LIN {X 0,Y 298.467,Z 190.307,A -85,B 0,C 180,E1 -16356.676,E2 -16356.676} C_VEL
LIN {X 0,Y 298.543,Z 190.3,A -85,B 0,C 180,E1 -16360.757,E2 -16360.757} C_VEL
LIN {X 0,Y 298.576,Z 190.293,A -85,B 0,C 180,E1 -16364.994,E2 -16364.994} C_VEL
LIN {X 0,Y 298.576,Z 190.292,A -85,B 0,C 180,E1 -16369.146,E2 -16369.146} C_VEL
LIN {X 0,Y 298.726,Z 190.273,A -85,B 0,C 180,E1 -16371.885,E2 -16371.885} C_VEL
LIN {X 0,Y 298.643,Z 190.285,A -85,B 0,C 180,E1 -16374.599,E2 -16374.599} C_VEL
LIN {X 0,Y 298.901,Z 190.252,A -85,B 0,C 180,E1 -16378.653,E2 -16378.653} C_VEL
LIN {X 0,Y 298.909,Z 190.249,A -85,B 0,C 180,E1 -16381.348,E2 -16381.348} C_VEL
LIN {X 0,Y 298.644,Z 190.283,A -85,B 0,C 180,E1 -16385.402,E2 -16385.402} C_VEL
LIN {X 0,Y 298.715,Z 190.277,A -85,B 0,C 180,E1 -16388.116,E2 -16388.116} C_VEL
LIN {X 0,Y 298.531,Z 190.298,A -85,B 0,C 180,E1 -16392.233,E2 -16392.233} C_VEL
LIN {X 0,Y 298.57,Z 190.292,A -85,B 0,C 180,E1 -16395.195,E2 -16395.195} C_VEL
LIN {X 0,Y 298.524,Z 190.3,A -85,B 0,C 180,E1 -16399.245,E2 -16399.245} C_VEL
LIN {X 0,Y 298.443,Z 190.31,A -85,B 0,C 180,E1 -16403.599,E2 -16403.599} C_VEL
LIN {X 0,Y 298.473,Z 190.303,A -85,B 0,C 180,E1 -16406.576,E2 -16406.576} C_VEL
LIN {X 0,Y 298.409,Z 190.313,A -85,B 0,C 180,E1 -16409.643,E2 -16409.643} C_VEL
LIN {X 0,Y 298.385,Z 190.317,A -85,B 0,C 180,E1 -16412.802,E2 -16412.802} C_VEL
LIN {X 0,Y 298.434,Z 190.312,A -85,B 0,C 180,E1 -16416.808,E2 -16416.808} C_VEL
LIN {X 0,Y 298.379,Z 190.318,A -85,B 0,C 180,E1 -16421.089,E2 -16421.089} C_VEL
LIN {X 0,Y 298.393,Z 190.316,A -85,B 0,C 180,E1 -16423.105,E2 -16423.105} C_VEL
LIN {X 0,Y 298.365,Z 190.321,A -85,B 0,C 180,E1 -16426.917,E2 -16426.917} C_VEL
LIN {X 0,Y 298.344,Z 190.416,A -85,B 0,C 180,E1 -16428.923,E2 -16428.923} C_VEL
LIN {X 0,Y 298.563,Z 193.304,A -85,B 0,C 180,E1 -16432.266,E2 -16432.266} C_VEL
LIN {X 0,Y 298.418,Z 196.385,A -85,B 0,C 180,E1 -16435.584,E2 -16435.584} C_VEL
LIN {X 0,Y 298.069,Z 199.435,A -85,B 0,C 180,E1 -16438.755,E2 -16438.755} C_VEL
LIN {X 0,Y 297.76,Z 203.535,A -85,B 0,C 180,E1 -16442.859,E2 -16442.859} C_VEL
LIN {X 0,Y 302.246,Z 218.03,A -85,B 0,C 180,E1 -16443.997,E2 -16443.997} C_VEL
LIN {X 0,Y 305.227,Z 230.394,A -85,B 0,C 180,E1 -16445.154,E2 -16445.154} C_VEL
LIN {X 0,Y 307.051,Z 240.7,A -85,B 0,C 180,E1 -16446.285,E2 -16446.285} C_VEL
LIN {X 0,Y 307.3,Z 244.849,A -85,B 0,C 180,E1 -16446.769,E2 -16446.769} C_VEL
LIN {X 0,Y 305.731,Z 255.792,A -85,B 0,C 180,E1 -16448.066,E2 -16448.066} C_VEL
LIN {X 0,Y 303.889,Z 266.643,A -85,B 0,C 180,E1 -16449.703,E2 -16449.703} C_VEL
LIN {X 0,Y 302.308,Z 275.446,A -85,B 0,C 180,E1 -16451.358,E2 -16451.358} C_VEL
LIN {X 0,Y 300.868,Z 282.972,A -85,B 0,C 180,E1 -16453.093,E2 -16453.093} C_VEL
LIN {X 0,Y 299.745,Z 289.831,A -85,B 0,C 180,E1 -16455.054,E2 -16455.054} C_VEL
LIN {X 0,Y 298.55,Z 295.506,A -85,B 0,C 180,E1 -16457.077,E2 -16457.077} C_VEL
LIN {X 0,Y 297.731,Z 299.967,A -85,B 0,C 180,E1 -16459.115,E2 -16459.115} C_VEL
LIN {X 0,Y 297.363,Z 302.317,A -85,B 0,C 180,E1 -16460.477,E2 -16460.477} C_VEL
LIN {X 0,Y 297.061,Z 304.239,A -85,B 0,C 180,E1 -16461.839,E2 -16461.839} C_VEL
LIN {X 0,Y 296.697,Z 306.572,A -85,B 0,C 180,E1 -16464.203,E2 -16464.203} C_VEL
LIN {X 0,Y 296.631,Z 307.466,A -85,B 0,C 180,E1 -16465.923,E2 -16465.923} C_VEL
LIN {X 0,Y 296.574,Z 307.752,A -85,B 0,C 180,E1 -16467.283,E2 -16467.283} C_VEL
LIN {X 0,Y 296.52,Z 307.658,A -85,B 0,C 180,E1 -16468.641,E2 -16468.641} C_VEL
LIN {X 0,Y 296.528,Z 307.138,A -85,B 0,C 180,E1 -16469.999,E2 -16469.999} C_VEL
LIN {X 0,Y 296.769,Z 304.924,A -85,B 0,C 180,E1 -16472.714,E2 -16472.714} C_VEL
LIN {X 0,Y 297.167,Z 302.172,A -85,B 0,C 180,E1 -16474.747,E2 -16474.747} C_VEL
LIN {X 0,Y 297.771,Z 297.516,A -85,B 0,C 180,E1 -16477.205,E2 -16477.205} C_VEL
LIN {X 0,Y 298.63,Z 291.646,A -85,B 0,C 180,E1 -16479.48,E2 -16479.48} C_VEL
LIN {X 0,Y 299.615,Z 285.031,A -85,B 0,C 180,E1 -16481.499,E2 -16481.499} C_VEL
LIN {X 0,Y 301.103,Z 276.811,A -85,B 0,C 180,E1 -16483.496,E2 -16483.496} C_VEL
LIN {X 0,Y 302.376,Z 268.381,A -85,B 0,C 180,E1 -16485.156,E2 -16485.156} C_VEL
LIN {X 0,Y 303.801,Z 257.965,A -85,B 0,C 180,E1 -16486.806,E2 -16486.806} C_VEL
LIN {X 0,Y 305.133,Z 249.054,A -85,B 0,C 180,E1 -16487.94,E2 -16487.94} C_VEL
LIN {X 0,Y 305.873,Z 241.537,A -85,B 0,C 180,E1 -16488.762,E2 -16488.762} C_VEL
LIN {X 0,Y 304.35,Z 230.406,A -85,B 0,C 180,E1 -16489.929,E2 -16489.929} C_VEL
LIN {X 0,Y 301.664,Z 218.168,A -85,B 0,C 180,E1 -16491.009,E2 -16491.009} C_VEL
LIN {X 0,Y 298.079,Z 205.668,A -85,B 0,C 180,E1 -16491.918,E2 -16491.918} C_VEL
LIN {X 0,Y 297.554,Z 203.452,A -85,B 0,C 180,E1 -16492.052,E2 -16492.052} C_VEL
LIN {X 0,Y 297.889,Z 199.089,A -85,B 0,C 180,E1 -16496.294,E2 -16496.294} C_VEL
LIN {X 0,Y 298.135,Z 195.735,A -85,B 0,C 180,E1 -16499.669,E2 -16499.669} C_VEL
LIN {X 0,Y 298.333,Z 192.716,A -85,B 0,C 180,E1 -16502.804,E2 -16502.804} C_VEL
LIN {X 0,Y 298.394,Z 191.172,A -85,B 0,C 180,E1 -16504.477,E2 -16504.477} C_VEL
LIN {X 0,Y 298.365,Z 190.322,A -85,B 0,C 180,E1 -16506.073,E2 -16506.073} C_VEL
LIN {X 0,Y 298.39,Z 190.319,A -85,B 0,C 180,E1 -16509.485,E2 -16509.485} C_VEL
LIN {X 0,Y 298.415,Z 190.315,A -85,B 0,C 180,E1 -16513.106,E2 -16513.106} C_VEL
LIN {X 0,Y 298.455,Z 190.309,A -85,B 0,C 180,E1 -16516.929,E2 -16516.929} C_VEL
LIN {X 0,Y 298.414,Z 190.316,A -85,B 0,C 180,E1 -16520.997,E2 -16520.997} C_VEL
LIN {X 0,Y 298.402,Z 190.312,A -85,B 0,C 180,E1 -16523.927,E2 -16523.927} C_VEL
LIN {X 0,Y 298.375,Z 190.315,A -85,B 0,C 180,E1 -16527.981,E2 -16527.981} C_VEL
LIN {X 0,Y 298.442,Z 190.307,A -85,B 0,C 180,E1 -16531.902,E2 -16531.902} C_VEL
LIN {X 0,Y 298.471,Z 190.303,A -85,B 0,C 180,E1 -16534.922,E2 -16534.922} C_VEL
LIN {X 0,Y 298.45,Z 190.298,A -85,B 0,C 180,E1 -16537.866,E2 -16537.866} C_VEL
LIN {X 0,Y 298.534,Z 190.29,A -85,B 0,C 180,E1 -16540.756,E2 -16540.756} C_VEL
LIN {X 0,Y 298.568,Z 190.292,A -85,B 0,C 180,E1 -16544.993,E2 -16544.993} C_VEL
LIN {X 0,Y 298.598,Z 190.283,A -85,B 0,C 180,E1 -16549.146,E2 -16549.146} C_VEL
LIN {X 0,Y 298.754,Z 190.271,A -85,B 0,C 180,E1 -16551.885,E2 -16551.885} C_VEL
LIN {X 0,Y 298.766,Z 190.266,A -85,B 0,C 180,E1 -16553.042,E2 -16553.042} C_VEL
LIN {X 0,Y 298.162,Z 190.346,A -85,B 0,C 180,E1 -16554.166,E2 -16554.166} C_VEL
LIN {X 0,Y 295.36,Z 190.695,A -85,B 0,C 180,E1 -16555.997,E2 -16555.997} C_VEL
LIN {X 0,Y 292.958,Z 190.991,A -85,B 0,C 180,E1 -16557.483,E2 -16557.483} C_VEL
LIN {X 0,Y 291.935,Z 191.118,A -85,B 0,C 180,E1 -16558.634,E2 -16558.634} C_VEL
LIN {X 0,Y 291.858,Z 191.126,A -85,B 0,C 180,E1 -16559.023,E2 -16559.023} C_VEL
LIN {X 0,Y 291.866,Z 191.129,A -85,B 0,C 180,E1 -16561.379,E2 -16561.379} C_VEL
LIN {X 0,Y 291.609,Z 191.163,A -85,B 0,C 180,E1 -16565.532,E2 -16565.532} C_VEL
LIN {X 0,Y 291.682,Z 191.15,A -85,B 0,C 180,E1 -16568.312,E2 -16568.312} C_VEL
LIN {X 0,Y 291.495,Z 191.174,A -85,B 0,C 180,E1 -16572.532,E2 -16572.532} C_VEL
LIN {X 0,Y 291.485,Z 191.179,A -85,B 0,C 180,E1 -16575.38,E2 -16575.38} C_VEL
LIN {X 0,Y 291.461,Z 191.178,A -85,B 0,C 180,E1 -16579.894,E2 -16579.894} C_VEL
LIN {X 0,Y 291.406,Z 191.185,A -85,B 0,C 180,E1 -16584.205,E2 -16584.205} C_VEL
LIN {X 0,Y 291.401,Z 191.186,A -85,B 0,C 180,E1 -16587.274,E2 -16587.274} C_VEL
LIN {X 0,Y 291.316,Z 191.192,A -85,B 0,C 180,E1 -16590.439,E2 -16590.439} C_VEL
LIN {X 0,Y 291.324,Z 191.194,A -85,B 0,C 180,E1 -16593.701,E2 -16593.701} C_VEL
LIN {X 0,Y 291.38,Z 191.189,A -85,B 0,C 180,E1 -16597.262,E2 -16597.262} C_VEL
LIN {X 0,Y 291.385,Z 191.191,A -85,B 0,C 180,E1 -16600.634,E2 -16600.634} C_VEL
LIN {X 0,Y 291.484,Z 191.352,A -85,B 0,C 180,E1 -16604.365,E2 -16604.365} C_VEL
LIN {X 0,Y 292.156,Z 195.534,A -85,B 0,C 180,E1 -16608.221,E2 -16608.221} C_VEL
LIN {X 0,Y 292.726,Z 199.162,A -85,B 0,C 180,E1 -16611.379,E2 -16611.379} C_VEL
LIN {X 0,Y 292.864,Z 201.277,A -85,B 0,C 180,E1 -16613.139,E2 -16613.139} C_VEL
LIN {X 0,Y 292.676,Z 204.438,A -85,B 0,C 180,E1 -16615.65,E2 -16615.65} C_VEL
LIN {X 0,Y 291.929,Z 209.681,A -85,B 0,C 180,E1 -16619.635,E2 -16619.635} C_VEL
LIN {X 0,Y 291.017,Z 215.923,A -85,B 0,C 180,E1 -16624.237,E2 -16624.237} C_VEL
LIN {X 0,Y 290.861,Z 217.67,A -85,B 0,C 180,E1 -16625.405,E2 -16625.405} C_VEL
LIN {X 0,Y 293.908,Z 230.878,A -85,B 0,C 180,E1 -16626.259,E2 -16626.259} C_VEL
LIN {X 0,Y 296.022,Z 243.414,A -85,B 0,C 180,E1 -16627.287,E2 -16627.287} C_VEL
LIN {X 0,Y 297.282,Z 255.41,A -85,B 0,C 180,E1 -16628.483,E2 -16628.483} C_VEL
LIN {X 0,Y 297.664,Z 263.572,A -85,B 0,C 180,E1 -16629.441,E2 -16629.441} C_VEL
LIN {X 0,Y 295.955,Z 275.139,A -85,B 0,C 180,E1 -16630.945,E2 -16630.945} C_VEL
LIN {X 0,Y 294.469,Z 284.874,A -85,B 0,C 180,E1 -16632.547,E2 -16632.547} C_VEL
LIN {X 0,Y 293.094,Z 293.699,A -85,B 0,C 180,E1 -16634.352,E2 -16634.352} C_VEL
LIN {X 0,Y 291.791,Z 301.858,A -85,B 0,C 180,E1 -16636.42,E2 -16636.42} C_VEL
LIN {X 0,Y 290.885,Z 307.407,A -85,B 0,C 180,E1 -16638.151,E2 -16638.151} C_VEL
LIN {X 0,Y 290.171,Z 312.836,A -85,B 0,C 180,E1 -16640.241,E2 -16640.241} C_VEL
LIN {X 0,Y 289.724,Z 317.078,A -85,B 0,C 180,E1 -16642.334,E2 -16642.334} C_VEL
LIN {X 0,Y 289.474,Z 320.363,A -85,B 0,C 180,E1 -16644.514,E2 -16644.514} C_VEL
LIN {X 0,Y 289.431,Z 321.835,A -85,B 0,C 180,E1 -16645.824,E2 -16645.824} C_VEL
LIN {X 0,Y 289.438,Z 322.994,A -85,B 0,C 180,E1 -16647.218,E2 -16647.218} C_VEL
LIN {X 0,Y 289.415,Z 323.716,A -85,B 0,C 180,E1 -16648.61,E2 -16648.61} C_VEL
LIN {X 0,Y 289.435,Z 324.052,A -85,B 0,C 180,E1 -16650.001,E2 -16650.001} C_VEL
LIN {X 0,Y 289.407,Z 324,A -85,B 0,C 180,E1 -16651.392,E2 -16651.392} C_VEL
LIN {X 0,Y 289.429,Z 323.552,A -85,B 0,C 180,E1 -16652.784,E2 -16652.784} C_VEL
LIN {X 0,Y 289.476,Z 321.389,A -85,B 0,C 180,E1 -16655.574,E2 -16655.574} C_VEL
LIN {X 0,Y 289.728,Z 318.686,A -85,B 0,C 180,E1 -16657.667,E2 -16657.667} C_VEL
LIN {X 0,Y 290.255,Z 314.97,A -85,B 0,C 180,E1 -16659.759,E2 -16659.759} C_VEL
LIN {X 0,Y 291.005,Z 310.143,A -85,B 0,C 180,E1 -16661.846,E2 -16661.846} C_VEL
LIN {X 0,Y 292.152,Z 304.062,A -85,B 0,C 180,E1 -16663.919,E2 -16663.919} C_VEL
LIN {X 0,Y 293.63,Z 296.509,A -85,B 0,C 180,E1 -16665.977,E2 -16665.977} C_VEL
LIN {X 0,Y 295.102,Z 288.16,A -85,B 0,C 180,E1 -16667.811,E2 -16667.811} C_VEL
LIN {X 0,Y 296.864,Z 278.345,A -85,B 0,C 180,E1 -16669.535,E2 -16669.535} C_VEL
LIN {X 0,Y 298.763,Z 267.709,A -85,B 0,C 180,E1 -16671.022,E2 -16671.022} C_VEL
LIN {X 0,Y 299.201,Z 263.555,A -85,B 0,C 180,E1 -16671.531,E2 -16671.531} C_VEL
LIN {X 0,Y 298.318,Z 252.514,A -85,B 0,C 180,E1 -16672.845,E2 -16672.845} C_VEL
LIN {X 0,Y 296.83,Z 241.889,A -85,B 0,C 180,E1 -16673.919,E2 -16673.919} C_VEL
LIN {X 0,Y 294.402,Z 229.74,A -85,B 0,C 180,E1 -16674.961,E2 -16674.961} C_VEL
LIN {X 0,Y 291.231,Z 217.803,A -85,B 0,C 180,E1 -16675.81,E2 -16675.81} C_VEL
LIN {X 0,Y 291.171,Z 217.363,A -85,B 0,C 180,E1 -16675.83,E2 -16675.83} C_VEL
LIN {X 0,Y 292.11,Z 211.302,A -85,B 0,C 180,E1 -16680.346,E2 -16680.346} C_VEL
LIN {X 0,Y 292.873,Z 206.162,A -85,B 0,C 180,E1 -16684.326,E2 -16684.326} C_VEL
LIN {X 0,Y 293.02,Z 202.084,A -85,B 0,C 180,E1 -16687.675,E2 -16687.675} C_VEL
LIN {X 0,Y 292.72,Z 198.923,A -85,B 0,C 180,E1 -16690.407,E2 -16690.407} C_VEL
LIN {X 0,Y 292.016,Z 194.786,A -85,B 0,C 180,E1 -16694.26,E2 -16694.26} C_VEL
LIN {X 0,Y 291.354,Z 191.198,A -85,B 0,C 180,E1 -16698.017,E2 -16698.017} C_VEL
LIN {X 0,Y 291.342,Z 191.196,A -85,B 0,C 180,E1 -16701.157,E2 -16701.157} C_VEL
LIN {X 0,Y 291.35,Z 191.195,A -85,B 0,C 180,E1 -16704.625,E2 -16704.625} C_VEL
LIN {X 0,Y 291.353,Z 191.194,A -85,B 0,C 180,E1 -16707.949,E2 -16707.949} C_VEL
LIN {X 0,Y 291.354,Z 191.196,A -85,B 0,C 180,E1 -16711.156,E2 -16711.156} C_VEL
LIN {X 0,Y 291.401,Z 191.185,A -85,B 0,C 180,E1 -16714.271,E2 -16714.271} C_VEL
LIN {X 0,Y 291.408,Z 191.186,A -85,B 0,C 180,E1 -16717.302,E2 -16717.302} C_VEL
LIN {X 0,Y 291.49,Z 191.175,A -85,B 0,C 180,E1 -16720.273,E2 -16720.273} C_VEL
LIN {X 0,Y 291.526,Z 191.174,A -85,B 0,C 180,E1 -16724.634,E2 -16724.634} C_VEL
LIN {X 0,Y 291.52,Z 191.172,A -85,B 0,C 180,E1 -16728.88,E2 -16728.88} C_VEL
LIN {X 0,Y 291.673,Z 191.151,A -85,B 0,C 180,E1 -16731.688,E2 -16731.688} C_VEL
LIN {X 0,Y 291.613,Z 191.161,A -85,B 0,C 180,E1 -16734.468,E2 -16734.468} C_VEL
LIN {X 0,Y 291.868,Z 191.129,A -85,B 0,C 180,E1 -16738.621,E2 -16738.621} C_VEL
LIN {X 0,Y 291.876,Z 191.125,A -85,B 0,C 180,E1 -16741.38,E2 -16741.38} C_VEL
LIN {X 0,Y 291.614,Z 191.16,A -85,B 0,C 180,E1 -16745.532,E2 -16745.532} C_VEL
LIN {X 0,Y 291.664,Z 191.153,A -85,B 0,C 180,E1 -16748.313,E2 -16748.313} C_VEL
LIN {X 0,Y 291.499,Z 191.173,A -85,B 0,C 180,E1 -16752.533,E2 -16752.533} C_VEL
LIN {X 0,Y 291.524,Z 191.171,A -85,B 0,C 180,E1 -16755.378,E2 -16755.378} C_VEL
LIN {X 0,Y 291.438,Z 191.183,A -85,B 0,C 180,E1 -16759.876,E2 -16759.876} C_VEL
LIN {X 0,Y 291.385,Z 191.186,A -85,B 0,C 180,E1 -16764.207,E2 -16764.207} C_VEL
LIN {X 0,Y 291.408,Z 191.188,A -85,B 0,C 180,E1 -16767.273,E2 -16767.273} C_VEL
LIN {X 0,Y 291.326,Z 191.194,A -85,B 0,C 180,E1 -16770.439,E2 -16770.439} C_VEL
LIN {X 0,Y 291.334,Z 191.194,A -85,B 0,C 180,E1 -16773.7,E2 -16773.7} C_VEL
LIN {X 0,Y 291.362,Z 191.191,A -85,B 0,C 180,E1 -16777.254,E2 -16777.254} C_VEL
LIN {X 0,Y 291.324,Z 191.197,A -85,B 0,C 180,E1 -16780.645,E2 -16780.645} C_VEL
LIN {X 0,Y 291.285,Z 191.202,A -85,B 0,C 180,E1 -16784.404,E2 -16784.404} C_VEL
LIN {X 0,Y 291.289,Z 191.203,A -85,B 0,C 180,E1 -16788.413,E2 -16788.413} C_VEL
LIN {X 0,Y 291.533,Z 193.453,A -85,B 0,C 180,E1 -16791.189,E2 -16791.189} C_VEL
LIN {X 0,Y 291.548,Z 195.003,A -85,B 0,C 180,E1 -16792.942,E2 -16792.942} C_VEL
LIN {X 0,Y 291.283,Z 198.076,A -85,B 0,C 180,E1 -16796.295,E2 -16796.295} C_VEL
LIN {X 0,Y 290.967,Z 201.142,A -85,B 0,C 180,E1 -16799.522,E2 -16799.522} C_VEL
LIN {X 0,Y 290.749,Z 203.759,A -85,B 0,C 180,E1 -16802.196,E2 -16802.196} C_VEL
LIN {X 0,Y 294.319,Z 214.776,A -85,B 0,C 180,E1 -16803.063,E2 -16803.063} C_VEL
LIN {X 0,Y 297.609,Z 227.072,A -85,B 0,C 180,E1 -16804.212,E2 -16804.212} C_VEL
LIN {X 0,Y 299.924,Z 239.037,A -85,B 0,C 180,E1 -16805.521,E2 -16805.521} C_VEL
LIN {X 0,Y 300.63,Z 245.942,A -85,B 0,C 180,E1 -16806.353,E2 -16806.353} C_VEL
LIN {X 0,Y 298.943,Z 256.985,A -85,B 0,C 180,E1 -16807.723,E2 -16807.723} C_VEL
LIN {X 0,Y 297.212,Z 266.692,A -85,B 0,C 180,E1 -16809.226,E2 -16809.226} C_VEL
LIN {X 0,Y 295.583,Z 275.52,A -85,B 0,C 180,E1 -16810.918,E2 -16810.918} C_VEL
LIN {X 0,Y 294.067,Z 283.067,A -85,B 0,C 180,E1 -16812.69,E2 -16812.69} C_VEL
LIN {X 0,Y 292.837,Z 289.948,A -85,B 0,C 180,E1 -16814.693,E2 -16814.693} C_VEL
LIN {X 0,Y 291.61,Z 295.642,A -85,B 0,C 180,E1 -16816.764,E2 -16816.764} C_VEL
LIN {X 0,Y 290.733,Z 300.118,A -85,B 0,C 180,E1 -16818.849,E2 -16818.849} C_VEL
LIN {X 0,Y 290.332,Z 302.475,A -85,B 0,C 180,E1 -16820.244,E2 -16820.244} C_VEL
LIN {X 0,Y 290.007,Z 304.403,A -85,B 0,C 180,E1 -16821.639,E2 -16821.639} C_VEL
LIN {X 0,Y 289.597,Z 306.896,A -85,B 0,C 180,E1 -16824.272,E2 -16824.272} C_VEL
LIN {X 0,Y 289.55,Z 307.654,A -85,B 0,C 180,E1 -16825.824,E2 -16825.824} C_VEL
LIN {X 0,Y 289.503,Z 307.946,A -85,B 0,C 180,E1 -16827.216,E2 -16827.216} C_VEL
LIN {X 0,Y 289.441,Z 307.86,A -85,B 0,C 180,E1 -16828.608,E2 -16828.608} C_VEL
LIN {X 0,Y 289.445,Z 307.351,A -85,B 0,C 180,E1 -16829.999,E2 -16829.999} C_VEL
LIN {X 0,Y 289.697,Z 305.149,A -85,B 0,C 180,E1 -16832.78,E2 -16832.78} C_VEL
LIN {X 0,Y 290.119,Z 302.41,A -85,B 0,C 180,E1 -16834.862,E2 -16834.862} C_VEL
LIN {X 0,Y 290.631,Z 298.666,A -85,B 0,C 180,E1 -16836.943,E2 -16836.943} C_VEL
LIN {X 0,Y 291.344,Z 293.809,A -85,B 0,C 180,E1 -16839.019,E2 -16839.019} C_VEL
LIN {X 0,Y 292.281,Z 287.695,A -85,B 0,C 180,E1 -16841.089,E2 -16841.089} C_VEL
LIN {X 0,Y 293.672,Z 280.075,A -85,B 0,C 180,E1 -16843.139,E2 -16843.139} C_VEL
LIN {X 0,Y 295.257,Z 270.503,A -85,B 0,C 180,E1 -16845.177,E2 -16845.177} C_VEL
LIN {X 0,Y 296.76,Z 260.627,A -85,B 0,C 180,E1 -16846.862,E2 -16846.862} C_VEL
LIN {X 0,Y 298.153,Z 250.883,A -85,B 0,C 180,E1 -16848.197,E2 -16848.197} C_VEL
LIN {X 0,Y 299.049,Z 243.545,A -85,B 0,C 180,E1 -16849.029,E2 -16849.029} C_VEL
LIN {X 0,Y 298.349,Z 236.105,A -85,B 0,C 180,E1 -16849.87,E2 -16849.87} C_VEL
LIN {X 0,Y 296.394,Z 225.434,A -85,B 0,C 180,E1 -16850.941,E2 -16850.941} C_VEL
LIN {X 0,Y 293.199,Z 212.867,A -85,B 0,C 180,E1 -16852,E2 -16852} C_VEL
LIN {X 0,Y 290.55,Z 203.62,A -85,B 0,C 180,E1 -16852.658,E2 -16852.658} C_VEL
LIN {X 0,Y 290.859,Z 199.679,A -85,B 0,C 180,E1 -16856.615,E2 -16856.615} C_VEL
LIN {X 0,Y 291.162,Z 195.954,A -85,B 0,C 180,E1 -16860.454,E2 -16860.454} C_VEL
LIN {X 0,Y 291.334,Z 192.925,A -85,B 0,C 180,E1 -16863.696,E2 -16863.696} C_VEL
LIN {X 0,Y 291.305,Z 191.439,A -85,B 0,C 180,E1 -16865.378,E2 -16865.378} C_VEL
LIN {X 0,Y 291.343,Z 191.198,A -85,B 0,C 180,E1 -16867.244,E2 -16867.244} C_VEL
LIN {X 0,Y 291.323,Z 191.196,A -85,B 0,C 180,E1 -16870.639,E2 -16870.639} C_VEL
LIN {X 0,Y 291.331,Z 191.195,A -85,B 0,C 180,E1 -16874.389,E2 -16874.389} C_VEL
LIN {X 0,Y 291.372,Z 191.189,A -85,B 0,C 180,E1 -16878.388,E2 -16878.388} C_VEL
LIN {X 0,Y 291.362,Z 191.193,A -85,B 0,C 180,E1 -16881.159,E2 -16881.159} C_VEL
LIN {X 0,Y 291.345,Z 191.194,A -85,B 0,C 180,E1 -16884.623,E2 -16884.623} C_VEL
LIN {X 0,Y 291.352,Z 191.19,A -85,B 0,C 180,E1 -16887.948,E2 -16887.948} C_VEL
LIN {X 0,Y 291.361,Z 191.19,A -85,B 0,C 180,E1 -16891.156,E2 -16891.156} C_VEL
LIN {X 0,Y 291.398,Z 191.187,A -85,B 0,C 180,E1 -16894.27,E2 -16894.27} C_VEL
LIN {X 0,Y 291.401,Z 191.174,A -85,B 0,C 180,E1 -16897.301,E2 -16897.301} C_VEL
LIN {X 0,Y 291.482,Z 191.16,A -85,B 0,C 180,E1 -16900.271,E2 -16900.271} C_VEL
LIN {X 0,Y 291.517,Z 191.172,A -85,B 0,C 180,E1 -16904.633,E2 -16904.633} C_VEL
LIN {X 0,Y 291.533,Z 191.163,A -85,B 0,C 180,E1 -16908.88,E2 -16908.88} C_VEL
LIN {X 0,Y 291.702,Z 191.148,A -85,B 0,C 180,E1 -16911.688,E2 -16911.688} C_VEL
LIN {X 0,Y 291.609,Z 191.158,A -85,B 0,C 180,E1 -16914.468,E2 -16914.468} C_VEL
LIN {X 0,Y 291.86,Z 191.127,A -85,B 0,C 180,E1 -16918.62,E2 -16918.62} C_VEL
LIN {X 0,Y 291.858,Z 191.126,A -85,B 0,C 180,E1 -16919.023,E2 -16919.023} C_VEL
LIN {X 0,Y 291.164,Z 191.216,A -85,B 0,C 180,E1 -16920.176,E2 -16920.176} C_VEL
LIN {X 0,Y 288.155,Z 191.591,A -85,B 0,C 180,E1 -16922.047,E2 -16922.047} C_VEL
LIN {X 0,Y 285.627,Z 191.908,A -85,B 0,C 180,E1 -16923.567,E2 -16923.567} C_VEL
LIN {X 0,Y 284.588,Z 192.033,A -85,B 0,C 180,E1 -16924.749,E2 -16924.749} C_VEL
LIN {X 0,Y 284.529,Z 192.041,A -85,B 0,C 180,E1 -16925.15,E2 -16925.15} C_VEL
LIN {X 0,Y 284.672,Z 192.024,A -85,B 0,C 180,E1 -16927.09,E2 -16927.09} C_VEL
LIN {X 0,Y 284.542,Z 192.041,A -85,B 0,C 180,E1 -16929.956,E2 -16929.956} C_VEL
LIN {X 0,Y 284.445,Z 192.051,A -85,B 0,C 180,E1 -16934.304,E2 -16934.304} C_VEL
LIN {X 0,Y 284.398,Z 192.06,A -85,B 0,C 180,E1 -16938.739,E2 -16938.739} C_VEL
LIN {X 0,Y 284.335,Z 192.066,A -85,B 0,C 180,E1 -16941.762,E2 -16941.762} C_VEL
LIN {X 0,Y 284.34,Z 192.068,A -85,B 0,C 180,E1 -16944.846,E2 -16944.846} C_VEL
LIN {X 0,Y 284.31,Z 192.068,A -85,B 0,C 180,E1 -16948.013,E2 -16948.013} C_VEL
LIN {X 0,Y 284.274,Z 192.07,A -85,B 0,C 180,E1 -16951.277,E2 -16951.277} C_VEL
LIN {X 0,Y 284.343,Z 192.065,A -85,B 0,C 180,E1 -16955.356,E2 -16955.356} C_VEL
LIN {X 0,Y 284.313,Z 192.071,A -85,B 0,C 180,E1 -16958.169,E2 -16958.169} C_VEL
LIN {X 0,Y 284.327,Z 192.07,A -85,B 0,C 180,E1 -16962.143,E2 -16962.143} C_VEL
LIN {X 0,Y 284.381,Z 192.07,A -85,B 0,C 180,E1 -16963.786,E2 -16963.786} C_VEL
LIN {X 0,Y 285.063,Z 196.148,A -85,B 0,C 180,E1 -16967.699,E2 -16967.699} C_VEL
LIN {X 0,Y 285.517,Z 198.928,A -85,B 0,C 180,E1 -16970.214,E2 -16970.214} C_VEL
LIN {X 0,Y 285.824,Z 202.11,A -85,B 0,C 180,E1 -16972.961,E2 -16972.961} C_VEL
LIN {X 0,Y 285.667,Z 205.267,A -85,B 0,C 180,E1 -16975.543,E2 -16975.543} C_VEL
LIN {X 0,Y 284.838,Z 210.638,A -85,B 0,C 180,E1 -16979.721,E2 -16979.721} C_VEL
LIN {X 0,Y 284.074,Z 215.694,A -85,B 0,C 180,E1 -16983.559,E2 -16983.559} C_VEL
LIN {X 0,Y 283.873,Z 217.305,A -85,B 0,C 180,E1 -16984.77,E2 -16984.77} C_VEL
LIN {X 0,Y 287.066,Z 230.901,A -85,B 0,C 180,E1 -16985.697,E2 -16985.697} C_VEL
LIN {X 0,Y 289.187,Z 243.352,A -85,B 0,C 180,E1 -16986.755,E2 -16986.755} C_VEL
LIN {X 0,Y 290.454,Z 255.674,A -85,B 0,C 180,E1 -16988.024,E2 -16988.024} C_VEL
LIN {X 0,Y 290.924,Z 263.193,A -85,B 0,C 180,E1 -16988.943,E2 -16988.943} C_VEL
LIN {X 0,Y 289.25,Z 274.797,A -85,B 0,C 180,E1 -16990.485,E2 -16990.485} C_VEL
LIN {X 0,Y 287.883,Z 283.112,A -85,B 0,C 180,E1 -16991.857,E2 -16991.857} C_VEL
LIN {X 0,Y 286.548,Z 291.888,A -85,B 0,C 180,E1 -16993.619,E2 -16993.619} C_VEL
LIN {X 0,Y 285.081,Z 300.345,A -85,B 0,C 180,E1 -16995.73,E2 -16995.73} C_VEL
LIN {X 0,Y 283.883,Z 307.145,A -85,B 0,C 180,E1 -16997.854,E2 -16997.854} C_VEL
LIN {X 0,Y 283.149,Z 312.588,A -85,B 0,C 180,E1 -16999.996,E2 -16999.996} C_VEL
LIN {X 0,Y 282.678,Z 316.842,A -85,B 0,C 180,E1 -17002.142,E2 -17002.142} C_VEL
LIN {X 0,Y 282.369,Z 320.431,A -85,B 0,C 180,E1 -17004.61,E2 -17004.61} C_VEL
LIN {X 0,Y 282.345,Z 322.783,A -85,B 0,C 180,E1 -17007.148,E2 -17007.148} C_VEL
LIN {X 0,Y 282.338,Z 323.512,A -85,B 0,C 180,E1 -17008.575,E2 -17008.575} C_VEL
LIN {X 0,Y 282.354,Z 323.852,A -85,B 0,C 180,E1 -17010.001,E2 -17010.001} C_VEL
LIN {X 0,Y 282.33,Z 323.805,A -85,B 0,C 180,E1 -17011.427,E2 -17011.427} C_VEL
LIN {X 0,Y 282.335,Z 323.365,A -85,B 0,C 180,E1 -17012.854,E2 -17012.854} C_VEL
LIN {X 0,Y 282.385,Z 321.213,A -85,B 0,C 180,E1 -17015.714,E2 -17015.714} C_VEL
LIN {X 0,Y 282.685,Z 318.521,A -85,B 0,C 180,E1 -17017.86,E2 -17017.86} C_VEL
LIN {X 0,Y 283.22,Z 314.815,A -85,B 0,C 180,E1 -17020.003,E2 -17020.003} C_VEL
LIN {X 0,Y 284.031,Z 310,A -85,B 0,C 180,E1 -17022.141,E2 -17022.141} C_VEL
LIN {X 0,Y 285.239,Z 303.932,A -85,B 0,C 180,E1 -17024.264,E2 -17024.264} C_VEL
LIN {X 0,Y 286.757,Z 296.393,A -85,B 0,C 180,E1 -17026.37,E2 -17026.37} C_VEL
LIN {X 0,Y 288.258,Z 288.423,A -85,B 0,C 180,E1 -17028.173,E2 -17028.173} C_VEL
LIN {X 0,Y 290.152,Z 278.279,A -85,B 0,C 180,E1 -17030.006,E2 -17030.006} C_VEL
LIN {X 0,Y 292.147,Z 267.67,A -85,B 0,C 180,E1 -17031.521,E2 -17031.521} C_VEL
LIN {X 0,Y 292.393,Z 263.533,A -85,B 0,C 180,E1 -17032.059,E2 -17032.059} C_VEL
LIN {X 0,Y 291.611,Z 253.19,A -85,B 0,C 180,E1 -17033.332,E2 -17033.332} C_VEL
LIN {X 0,Y 289.912,Z 240.989,A -85,B 0,C 180,E1 -17034.611,E2 -17034.611} C_VEL
LIN {X 0,Y 287.221,Z 228.353,A -85,B 0,C 180,E1 -17035.72,E2 -17035.72} C_VEL
LIN {X 0,Y 284.247,Z 217.152,A -85,B 0,C 180,E1 -17036.545,E2 -17036.545} C_VEL
LIN {X 0,Y 285.064,Z 212.15,A -85,B 0,C 180,E1 -17040.357,E2 -17040.357} C_VEL
LIN {X 0,Y 285.845,Z 207.016,A -85,B 0,C 180,E1 -17044.435,E2 -17044.435} C_VEL
LIN {X 0,Y 286.032,Z 203.954,A -85,B 0,C 180,E1 -17047.01,E2 -17047.01} C_VEL
LIN {X 0,Y 285.743,Z 200.215,A -85,B 0,C 180,E1 -17050.319,E2 -17050.319} C_VEL
LIN {X 0,Y 285.166,Z 196.71,A -85,B 0,C 180,E1 -17053.633,E2 -17053.633} C_VEL
LIN {X 0,Y 284.386,Z 192.568,A -85,B 0,C 180,E1 -17057.846,E2 -17057.846} C_VEL
LIN {X 0,Y 284.284,Z 192.076,A -85,B 0,C 180,E1 -17058.601,E2 -17058.601} C_VEL
LIN {X 0,Y 284.311,Z 192.07,A -85,B 0,C 180,E1 -17062.277,E2 -17062.277} C_VEL
LIN {X 0,Y 284.297,Z 192.076,A -85,B 0,C 180,E1 -17065.349,E2 -17065.349} C_VEL
LIN {X 0,Y 284.275,Z 192.077,A -85,B 0,C 180,E1 -17068.723,E2 -17068.723} C_VEL
LIN {X 0,Y 284.378,Z 192.063,A -85,B 0,C 180,E1 -17072.828,E2 -17072.828} C_VEL
LIN {X 0,Y 284.37,Z 192.064,A -85,B 0,C 180,E1 -17076.707,E2 -17076.707} C_VEL
LIN {X 0,Y 284.418,Z 192.055,A -85,B 0,C 180,E1 -17079.873,E2 -17079.873} C_VEL
LIN {X 0,Y 284.463,Z 192.052,A -85,B 0,C 180,E1 -17084.469,E2 -17084.469} C_VEL
LIN {X 0,Y 284.472,Z 192.052,A -85,B 0,C 180,E1 -17088.601,E2 -17088.601} C_VEL
LIN {X 0,Y 284.624,Z 192.029,A -85,B 0,C 180,E1 -17091.48,E2 -17091.48} C_VEL
LIN {X 0,Y 284.583,Z 192.038,A -85,B 0,C 180,E1 -17094.331,E2 -17094.331} C_VEL
LIN {X 0,Y 284.834,Z 192.005,A -85,B 0,C 180,E1 -17098.586,E2 -17098.586} C_VEL
LIN {X 0,Y 284.842,Z 192.002,A -85,B 0,C 180,E1 -17101.414,E2 -17101.414} C_VEL
LIN {X 0,Y 284.624,Z 192.027,A -85,B 0,C 180,E1 -17106.681,E2 -17106.681} C_VEL
LIN {X 0,Y 284.498,Z 192.048,A -85,B 0,C 180,E1 -17109.958,E2 -17109.958} C_VEL
LIN {X 0,Y 284.462,Z 192.049,A -85,B 0,C 180,E1 -17114.304,E2 -17114.304} C_VEL
LIN {X 0,Y 284.411,Z 192.057,A -85,B 0,C 180,E1 -17117.25,E2 -17117.25} C_VEL
LIN {X 0,Y 284.366,Z 192.062,A -85,B 0,C 180,E1 -17120.244,E2 -17120.244} C_VEL
LIN {X 0,Y 284.355,Z 192.063,A -85,B 0,C 180,E1 -17123.876,E2 -17123.876} C_VEL
LIN {X 0,Y 284.384,Z 192.062,A -85,B 0,C 180,E1 -17127.174,E2 -17127.174} C_VEL
LIN {X 0,Y 284.284,Z 192.075,A -85,B 0,C 180,E1 -17131.276,E2 -17131.276} C_VEL
LIN {X 0,Y 284.331,Z 192.069,A -85,B 0,C 180,E1 -17135.349,E2 -17135.349} C_VEL
LIN {X 0,Y 284.299,Z 192.07,A -85,B 0,C 180,E1 -17138.172,E2 -17138.172} C_VEL
LIN {X 0,Y 284.262,Z 192.074,A -85,B 0,C 180,E1 -17142.126,E2 -17142.126} C_VEL
LIN {X 0,Y 284.232,Z 192.081,A -85,B 0,C 180,E1 -17146.187,E2 -17146.187} C_VEL
LIN {X 0,Y 284.236,Z 192.081,A -85,B 0,C 180,E1 -17148.12,E2 -17148.12} C_VEL
LIN {X 0,Y 284.447,Z 193.606,A -85,B 0,C 180,E1 -17150.031,E2 -17150.031} C_VEL
LIN {X 0,Y 284.532,Z 195.458,A -85,B 0,C 180,E1 -17152.225,E2 -17152.225} C_VEL
LIN {X 0,Y 284.337,Z 198.246,A -85,B 0,C 180,E1 -17155.356,E2 -17155.356} C_VEL
LIN {X 0,Y 284.016,Z 201.326,A -85,B 0,C 180,E1 -17158.693,E2 -17158.693} C_VEL
LIN {X 0,Y 283.777,Z 203.946,A -85,B 0,C 180,E1 -17161.463,E2 -17161.463} C_VEL
LIN {X 0,Y 285.69,Z 209.796,A -85,B 0,C 180,E1 -17161.939,E2 -17161.939} C_VEL
LIN {X 0,Y 289.595,Z 222.519,A -85,B 0,C 180,E1 -17163.109,E2 -17163.109} C_VEL
LIN {X 0,Y 292.212,Z 234.223,A -85,B 0,C 180,E1 -17164.348,E2 -17164.348} C_VEL
LIN {X 0,Y 293.963,Z 245.479,A -85,B 0,C 180,E1 -17165.733,E2 -17165.733} C_VEL
LIN {X 0,Y 292.96,Z 253.243,A -85,B 0,C 180,E1 -17166.683,E2 -17166.683} C_VEL
LIN {X 0,Y 291.162,Z 263.722,A -85,B 0,C 180,E1 -17168.216,E2 -17168.216} C_VEL
LIN {X 0,Y 289.564,Z 272.278,A -85,B 0,C 180,E1 -17169.766,E2 -17169.766} C_VEL
LIN {X 0,Y 287.927,Z 280.156,A -85,B 0,C 180,E1 -17171.5,E2 -17171.5} C_VEL
LIN {X 0,Y 286.256,Z 287.917,A -85,B 0,C 180,E1 -17173.625,E2 -17173.625} C_VEL
LIN {X 0,Y 285.141,Z 293.992,A -85,B 0,C 180,E1 -17175.731,E2 -17175.731} C_VEL
LIN {X 0,Y 283.984,Z 298.875,A -85,B 0,C 180,E1 -17177.857,E2 -17177.857} C_VEL
LIN {X 0,Y 283.314,Z 302.632,A -85,B 0,C 180,E1 -17180,E2 -17180} C_VEL
LIN {X 0,Y 282.953,Z 304.568,A -85,B 0,C 180,E1 -17181.429,E2 -17181.429} C_VEL
LIN {X 0,Y 282.682,Z 306.091,A -85,B 0,C 180,E1 -17182.859,E2 -17182.859} C_VEL
LIN {X 0,Y 282.526,Z 307.167,A -85,B 0,C 180,E1 -17184.289,E2 -17184.289} C_VEL
LIN {X 0,Y 282.433,Z 308.14,A -85,B 0,C 180,E1 -17187.147,E2 -17187.147} C_VEL
LIN {X 0,Y 282.364,Z 308.061,A -85,B 0,C 180,E1 -17188.573,E2 -17188.573} C_VEL
LIN {X 0,Y 282.365,Z 307.563,A -85,B 0,C 180,E1 -17189.999,E2 -17189.999} C_VEL
LIN {X 0,Y 282.628,Z 305.374,A -85,B 0,C 180,E1 -17192.85,E2 -17192.85} C_VEL
LIN {X 0,Y 283.071,Z 302.647,A -85,B 0,C 180,E1 -17194.984,E2 -17194.984} C_VEL
LIN {X 0,Y 283.577,Z 298.918,A -85,B 0,C 180,E1 -17197.117,E2 -17197.117} C_VEL
LIN {X 0,Y 284.334,Z 294.076,A -85,B 0,C 180,E1 -17199.244,E2 -17199.244} C_VEL
LIN {X 0,Y 285.315,Z 287.978,A -85,B 0,C 180,E1 -17201.363,E2 -17201.363} C_VEL
LIN {X 0,Y 286.79,Z 280.382,A -85,B 0,C 180,E1 -17203.46,E2 -17203.46} C_VEL
LIN {X 0,Y 288.432,Z 270.835,A -85,B 0,C 180,E1 -17205.545,E2 -17205.545} C_VEL
LIN {X 0,Y 289.979,Z 260.987,A -85,B 0,C 180,E1 -17207.269,E2 -17207.269} C_VEL
LIN {X 0,Y 291.425,Z 251.36,A -85,B 0,C 180,E1 -17208.622,E2 -17208.622} C_VEL
LIN {X 0,Y 292.355,Z 243.333,A -85,B 0,C 180,E1 -17209.558,E2 -17209.558} C_VEL
LIN {X 0,Y 290.773,Z 232.018,A -85,B 0,C 180,E1 -17210.851,E2 -17210.851} C_VEL
LIN {X 0,Y 288.376,Z 220.872,A -85,B 0,C 180,E1 -17211.938,E2 -17211.938} C_VEL
LIN {X 0,Y 284.796,Z 208.325,A -85,B 0,C 180,E1 -17212.961,E2 -17212.961} C_VEL
LIN {X 0,Y 283.549,Z 203.835,A -85,B 0,C 180,E1 -17213.278,E2 -17213.278} C_VEL
LIN {X 0,Y 283.823,Z 200.244,A -85,B 0,C 180,E1 -17216.945,E2 -17216.945} C_VEL
LIN {X 0,Y 284.1,Z 197.348,A -85,B 0,C 180,E1 -17220.022,E2 -17220.022} C_VEL
LIN {X 0,Y 284.289,Z 194.648,A -85,B 0,C 180,E1 -17222.944,E2 -17222.944} C_VEL
LIN {X 0,Y 284.295,Z 192.544,A -85,B 0,C 180,E1 -17225.334,E2 -17225.334} C_VEL
LIN {X 0,Y 284.259,Z 192.08,A -85,B 0,C 180,E1 -17226.393,E2 -17226.393} C_VEL
LIN {X 0,Y 284.296,Z 192.072,A -85,B 0,C 180,E1 -17229.992,E2 -17229.992} C_VEL
LIN {X 0,Y 284.283,Z 192.073,A -85,B 0,C 180,E1 -17234.197,E2 -17234.197} C_VEL
LIN {X 0,Y 284.324,Z 192.067,A -85,B 0,C 180,E1 -17238.133,E2 -17238.133} C_VEL
LIN {X 0,Y 284.324,Z 192.067,A -85,B 0,C 180,E1 -17242.271,E2 -17242.271} C_VEL
LIN {X 0,Y 284.292,Z 192.072,A -85,B 0,C 180,E1 -17245.348,E2 -17245.348} C_VEL
LIN {X 0,Y 284.276,Z 192.075,A -85,B 0,C 180,E1 -17248.723,E2 -17248.723} C_VEL
LIN {X 0,Y 284.376,Z 192.063,A -85,B 0,C 180,E1 -17252.825,E2 -17252.825} C_VEL
LIN {X 0,Y 284.362,Z 192.053,A -85,B 0,C 180,E1 -17256.706,E2 -17256.706} C_VEL
LIN {X 0,Y 284.41,Z 192.036,A -85,B 0,C 180,E1 -17259.872,E2 -17259.872} C_VEL
LIN {X 0,Y 284.455,Z 192.053,A -85,B 0,C 180,E1 -17264.468,E2 -17264.468} C_VEL
LIN {X 0,Y 284.495,Z 192.04,A -85,B 0,C 180,E1 -17268.601,E2 -17268.601} C_VEL
LIN {X 0,Y 284.651,Z 192.025,A -85,B 0,C 180,E1 -17271.481,E2 -17271.481} C_VEL
LIN {X 0,Y 284.58,Z 192.034,A -85,B 0,C 180,E1 -17274.33,E2 -17274.33} C_VEL
LIN {X 0,Y 284.827,Z 192.003,A -85,B 0,C 180,E1 -17278.586,E2 -17278.586} C_VEL
LIN {X 0,Y 284.833,Z 192.005,A -85,B 0,C 180,E1 -17281.414,E2 -17281.414} C_VEL
LIN {X 0,Y 284.529,Z 192.041,A -85,B 0,C 180,E1 -17285.15,E2 -17285.15} C_VEL
LIN {X 0,Y 283.918,Z 192.12,A -85,B 0,C 180,E1 -17286.333,E2 -17286.333} C_VEL
LIN {X 0,Y 281.044,Z 192.475,A -85,B 0,C 180,E1 -17288.259,E2 -17288.259} C_VEL
LIN {X 0,Y 278.564,Z 192.786,A -85,B 0,C 180,E1 -17289.824,E2 -17289.824} C_VEL
LIN {X 0,Y 277.496,Z 192.92,A -85,B 0,C 180,E1 -17291.039,E2 -17291.039} C_VEL
LIN {X 0,Y 277.409,Z 192.929,A -85,B 0,C 180,E1 -17291.45,E2 -17291.45} C_VEL
LIN {X 0,Y 277.393,Z 192.932,A -85,B 0,C 180,E1 -17295.704,E2 -17295.704} C_VEL
LIN {X 0,Y 277.352,Z 192.936,A -85,B 0,C 180,E1 -17300.367,E2 -17300.367} C_VEL
LIN {X 0,Y 277.312,Z 192.94,A -85,B 0,C 180,E1 -17304.178,E2 -17304.178} C_VEL
LIN {X 0,Y 277.305,Z 192.941,A -85,B 0,C 180,E1 -17307.507,E2 -17307.507} C_VEL
LIN {X 0,Y 277.253,Z 192.942,A -85,B 0,C 180,E1 -17310.484,E2 -17310.484} C_VEL
LIN {X 0,Y 277.235,Z 192.949,A -85,B 0,C 180,E1 -17313.897,E2 -17313.897} C_VEL
LIN {X 0,Y 277.268,Z 192.946,A -85,B 0,C 180,E1 -17317.469,E2 -17317.469} C_VEL
LIN {X 0,Y 277.25,Z 192.95,A -85,B 0,C 180,E1 -17321.229,E2 -17321.229} C_VEL
LIN {X 0,Y 277.342,Z 193.015,A -85,B 0,C 180,E1 -17323.422,E2 -17323.422} C_VEL
LIN {X 0,Y 277.976,Z 196.793,A -85,B 0,C 180,E1 -17327.155,E2 -17327.155} C_VEL
LIN {X 0,Y 278.585,Z 200.823,A -85,B 0,C 180,E1 -17330.904,E2 -17330.904} C_VEL
LIN {X 0,Y 278.777,Z 204.123,A -85,B 0,C 180,E1 -17333.777,E2 -17333.777} C_VEL
LIN {X 0,Y 278.432,Z 207.309,A -85,B 0,C 180,E1 -17336.404,E2 -17336.404} C_VEL
LIN {X 0,Y 277.606,Z 212.36,A -85,B 0,C 180,E1 -17340.421,E2 -17340.421} C_VEL
LIN {X 0,Y 276.884,Z 217.101,A -85,B 0,C 180,E1 -17344.113,E2 -17344.113} C_VEL
LIN {X 0,Y 280.195,Z 230.818,A -85,B 0,C 180,E1 -17345.095,E2 -17345.095} C_VEL
LIN {X 0,Y 282.349,Z 243.629,A -85,B 0,C 180,E1 -17346.224,E2 -17346.224} C_VEL
LIN {X 0,Y 283.545,Z 254.802,A -85,B 0,C 180,E1 -17347.413,E2 -17347.413} C_VEL
LIN {X 0,Y 284.12,Z 264.251,A -85,B 0,C 180,E1 -17348.604,E2 -17348.604} C_VEL
LIN {X 0,Y 282.551,Z 274.452,A -85,B 0,C 180,E1 -17350.003,E2 -17350.003} C_VEL
LIN {X 0,Y 281.11,Z 282.848,A -85,B 0,C 180,E1 -17351.415,E2 -17351.415} C_VEL
LIN {X 0,Y 279.725,Z 291.588,A -85,B 0,C 180,E1 -17353.208,E2 -17353.208} C_VEL
LIN {X 0,Y 278.438,Z 298.797,A -85,B 0,C 180,E1 -17355.008,E2 -17355.008} C_VEL
LIN {X 0,Y 277.086,Z 305.869,A -85,B 0,C 180,E1 -17357.179,E2 -17357.179} C_VEL
LIN {X 0,Y 276.139,Z 312.34,A -85,B 0,C 180,E1 -17359.739,E2 -17359.739} C_VEL
LIN {X 0,Y 275.605,Z 316.605,A -85,B 0,C 180,E1 -17361.939,E2 -17361.939} C_VEL
LIN {X 0,Y 275.302,Z 319.8,A -85,B 0,C 180,E1 -17364.141,E2 -17364.141} C_VEL
LIN {X 0,Y 275.248,Z 321.394,A -85,B 0,C 180,E1 -17365.608,E2 -17365.608} C_VEL
LIN {X 0,Y 275.255,Z 322.572,A -85,B 0,C 180,E1 -17367.074,E2 -17367.074} C_VEL
LIN {X 0,Y 275.262,Z 323.307,A -85,B 0,C 180,E1 -17368.538,E2 -17368.538} C_VEL
LIN {X 0,Y 275.276,Z 323.653,A -85,B 0,C 180,E1 -17370.001,E2 -17370.001} C_VEL
LIN {X 0,Y 275.255,Z 323.611,A -85,B 0,C 180,E1 -17371.464,E2 -17371.464} C_VEL
LIN {X 0,Y 275.244,Z 323.177,A -85,B 0,C 180,E1 -17372.928,E2 -17372.928} C_VEL
LIN {X 0,Y 275.299,Z 321.037,A -85,B 0,C 180,E1 -17375.861,E2 -17375.861} C_VEL
LIN {X 0,Y 275.616,Z 318.355,A -85,B 0,C 180,E1 -17378.062,E2 -17378.062} C_VEL
LIN {X 0,Y 276.208,Z 314.661,A -85,B 0,C 180,E1 -17380.26,E2 -17380.26} C_VEL
LIN {X 0,Y 277.047,Z 309.857,A -85,B 0,C 180,E1 -17382.452,E2 -17382.452} C_VEL
LIN {X 0,Y 278.609,Z 302.684,A -85,B 0,C 180,E1 -17384.984,E2 -17384.984} C_VEL
LIN {X 0,Y 280.238,Z 294.852,A -85,B 0,C 180,E1 -17387.138,E2 -17387.138} C_VEL
LIN {X 0,Y 281.785,Z 286.87,A -85,B 0,C 180,E1 -17388.919,E2 -17388.919} C_VEL
LIN {X 0,Y 283.699,Z 277.143,A -85,B 0,C 180,E1 -17390.671,E2 -17390.671} C_VEL
LIN {X 0,Y 285.701,Z 266.338,A -85,B 0,C 180,E1 -17392.222,E2 -17392.222} C_VEL
LIN {X 0,Y 285.192,Z 256.761,A -85,B 0,C 180,E1 -17393.495,E2 -17393.495} C_VEL
LIN {X 0,Y 283.928,Z 246.122,A -85,B 0,C 180,E1 -17394.723,E2 -17394.723} C_VEL
LIN {X 0,Y 281.673,Z 233.669,A -85,B 0,C 180,E1 -17395.941,E2 -17395.941} C_VEL
LIN {X 0,Y 278.159,Z 220.165,A -85,B 0,C 180,E1 -17397.058,E2 -17397.058} C_VEL
LIN {X 0,Y 277.302,Z 216.932,A -85,B 0,C 180,E1 -17397.293,E2 -17397.293} C_VEL
LIN {X 0,Y 278.094,Z 212.533,A -85,B 0,C 180,E1 -17400.768,E2 -17400.768} C_VEL
LIN {X 0,Y 278.827,Z 207.894,A -85,B 0,C 180,E1 -17404.548,E2 -17404.548} C_VEL
LIN {X 0,Y 279.02,Z 204.833,A -85,B 0,C 180,E1 -17407.192,E2 -17407.192} C_VEL
LIN {X 0,Y 278.636,Z 200.713,A -85,B 0,C 180,E1 -17410.978,E2 -17410.978} C_VEL
LIN {X 0,Y 277.933,Z 196.693,A -85,B 0,C 180,E1 -17414.926,E2 -17414.926} C_VEL
LIN {X 0,Y 277.24,Z 192.954,A -85,B 0,C 180,E1 -17418.984,E2 -17418.984} C_VEL
LIN {X 0,Y 277.256,Z 192.949,A -85,B 0,C 180,E1 -17422.529,E2 -17422.529} C_VEL
LIN {X 0,Y 277.235,Z 192.953,A -85,B 0,C 180,E1 -17426.103,E2 -17426.103} C_VEL
LIN {X 0,Y 277.251,Z 192.952,A -85,B 0,C 180,E1 -17429.537,E2 -17429.537} C_VEL
LIN {X 0,Y 277.339,Z 192.94,A -85,B 0,C 180,E1 -17432.862,E2 -17432.862} C_VEL
LIN {X 0,Y 277.331,Z 192.938,A -85,B 0,C 180,E1 -17436.08,E2 -17436.08} C_VEL
LIN {X 0,Y 277.357,Z 192.938,A -85,B 0,C 180,E1 -17440.767,E2 -17440.767} C_VEL
LIN {X 0,Y 277.412,Z 192.928,A -85,B 0,C 180,E1 -17445.325,E2 -17445.325} C_VEL
LIN {X 0,Y 277.446,Z 192.923,A -85,B 0,C 180,E1 -17449.787,E2 -17449.787} C_VEL
LIN {X 0,Y 277.627,Z 192.903,A -85,B 0,C 180,E1 -17452.729,E2 -17452.729} C_VEL
LIN {X 0,Y 277.801,Z 192.882,A -85,B 0,C 180,E1 -17458.551,E2 -17458.551} C_VEL
LIN {X 0,Y 277.809,Z 192.878,A -85,B 0,C 180,E1 -17461.45,E2 -17461.45} C_VEL
LIN {X 0,Y 277.572,Z 192.906,A -85,B 0,C 180,E1 -17466.699,E2 -17466.699} C_VEL
LIN {X 0,Y 277.55,Z 192.91,A -85,B 0,C 180,E1 -17469.073,E2 -17469.073} C_VEL
LIN {X 0,Y 277.397,Z 192.93,A -85,B 0,C 180,E1 -17473.181,E2 -17473.181} C_VEL
LIN {X 0,Y 277.388,Z 192.932,A -85,B 0,C 180,E1 -17476.183,E2 -17476.183} C_VEL
LIN {X 0,Y 277.333,Z 192.938,A -85,B 0,C 180,E1 -17480.351,E2 -17480.351} C_VEL
LIN {X 0,Y 277.305,Z 192.94,A -85,B 0,C 180,E1 -17484.17,E2 -17484.17} C_VEL
LIN {X 0,Y 277.313,Z 192.943,A -85,B 0,C 180,E1 -17487.506,E2 -17487.506} C_VEL
LIN {X 0,Y 277.263,Z 192.946,A -85,B 0,C 180,E1 -17490.483,E2 -17490.483} C_VEL
LIN {X 0,Y 277.238,Z 192.95,A -85,B 0,C 180,E1 -17493.898,E2 -17493.898} C_VEL
LIN {X 0,Y 277.255,Z 192.948,A -85,B 0,C 180,E1 -17497.472,E2 -17497.472} C_VEL
LIN {X 0,Y 277.202,Z 192.955,A -85,B 0,C 180,E1 -17501.239,E2 -17501.239} C_VEL
LIN {X 0,Y 277.189,Z 192.959,A -85,B 0,C 180,E1 -17505.23,E2 -17505.23} C_VEL
LIN {X 0,Y 277.187,Z 192.959,A -85,B 0,C 180,E1 -17507.332,E2 -17507.332} C_VEL
LIN {X 0,Y 277.349,Z 194.328,A -85,B 0,C 180,E1 -17509.482,E2 -17509.482} C_VEL
LIN {X 0,Y 277.498,Z 196.848,A -85,B 0,C 180,E1 -17512.569,E2 -17512.569} C_VEL
LIN {X 0,Y 277.205,Z 199.966,A -85,B 0,C 180,E1 -17516.1,E2 -17516.1} C_VEL
LIN {X 0,Y 276.81,Z 203.997,A -85,B 0,C 180,E1 -17520.534,E2 -17520.534} C_VEL
LIN {X 0,Y 276.807,Z 204.171,A -85,B 0,C 180,E1 -17520.719,E2 -17520.719} C_VEL
LIN {X 0,Y 278.655,Z 209.899,A -85,B 0,C 180,E1 -17521.194,E2 -17521.194} C_VEL
LIN {X 0,Y 282.357,Z 221.611,A -85,B 0,C 180,E1 -17522.309,E2 -17522.309} C_VEL
LIN {X 0,Y 285.109,Z 233.013,A -85,B 0,C 180,E1 -17523.552,E2 -17523.552} C_VEL
LIN {X 0,Y 287.003,Z 244.285,A -85,B 0,C 180,E1 -17524.965,E2 -17524.965} C_VEL
LIN {X 0,Y 287.325,Z 247.732,A -85,B 0,C 180,E1 -17525.43,E2 -17525.43} C_VEL
LIN {X 0,Y 285.357,Z 259.371,A -85,B 0,C 180,E1 -17526.985,E2 -17526.985} C_VEL
LIN {X 0,Y 283.565,Z 268.742,A -85,B 0,C 180,E1 -17528.558,E2 -17528.558} C_VEL
LIN {X 0,Y 281.803,Z 277.274,A -85,B 0,C 180,E1 -17530.326,E2 -17530.326} C_VEL
LIN {X 0,Y 279.945,Z 285.554,A -85,B 0,C 180,E1 -17532.467,E2 -17532.467} C_VEL
LIN {X 0,Y 278.666,Z 292.212,A -85,B 0,C 180,E1 -17534.644,E2 -17534.644} C_VEL
LIN {X 0,Y 277.325,Z 297.523,A -85,B 0,C 180,E1 -17536.816,E2 -17536.816} C_VEL
LIN {X 0,Y 276.514,Z 301.655,A -85,B 0,C 180,E1 -17539.011,E2 -17539.011} C_VEL
LIN {X 0,Y 275.92,Z 304.732,A -85,B 0,C 180,E1 -17541.209,E2 -17541.209} C_VEL
LIN {X 0,Y 275.619,Z 306.262,A -85,B 0,C 180,E1 -17542.675,E2 -17542.675} C_VEL
LIN {X 0,Y 275.44,Z 307.455,A -85,B 0,C 180,E1 -17544.336,E2 -17544.336} C_VEL
LIN {X 0,Y 275.341,Z 308.335,A -85,B 0,C 180,E1 -17547.073,E2 -17547.073} C_VEL
LIN {X 0,Y 275.29,Z 308.262,A -85,B 0,C 180,E1 -17548.536,E2 -17548.536} C_VEL
LIN {X 0,Y 275.287,Z 307.776,A -85,B 0,C 180,E1 -17549.999,E2 -17549.999} C_VEL
LIN {X 0,Y 275.561,Z 305.598,A -85,B 0,C 180,E1 -17552.923,E2 -17552.923} C_VEL
LIN {X 0,Y 276.026,Z 302.884,A -85,B 0,C 180,E1 -17555.111,E2 -17555.111} C_VEL
LIN {X 0,Y 276.53,Z 299.17,A -85,B 0,C 180,E1 -17557.299,E2 -17557.299} C_VEL
LIN {X 0,Y 277.329,Z 294.342,A -85,B 0,C 180,E1 -17559.479,E2 -17559.479} C_VEL
LIN {X 0,Y 278.375,Z 288.259,A -85,B 0,C 180,E1 -17561.65,E2 -17561.65} C_VEL
LIN {X 0,Y 279.914,Z 280.686,A -85,B 0,C 180,E1 -17563.797,E2 -17563.797} C_VEL
LIN {X 0,Y 281.624,Z 271.166,A -85,B 0,C 180,E1 -17565.931,E2 -17565.931} C_VEL
LIN {X 0,Y 283.238,Z 261.346,A -85,B 0,C 180,E1 -17567.693,E2 -17567.693} C_VEL
LIN {X 0,Y 284.705,Z 251.871,A -85,B 0,C 180,E1 -17569.062,E2 -17569.062} C_VEL
LIN {X 0,Y 285.604,Z 244.333,A -85,B 0,C 180,E1 -17569.972,E2 -17569.972} C_VEL
LIN {X 0,Y 284.007,Z 232.844,A -85,B 0,C 180,E1 -17571.341,E2 -17571.341} C_VEL
LIN {X 0,Y 281.489,Z 221.379,A -85,B 0,C 180,E1 -17572.512,E2 -17572.512} C_VEL
LIN {X 0,Y 278.019,Z 208.989,A -85,B 0,C 180,E1 -17573.565,E2 -17573.565} C_VEL
LIN {X 0,Y 276.529,Z 204.03,A -85,B 0,C 180,E1 -17573.929,E2 -17573.929} C_VEL
LIN {X 0,Y 276.817,Z 200.847,A -85,B 0,C 180,E1 -17577.3,E2 -17577.3} C_VEL
LIN {X 0,Y 277.091,Z 197.898,A -85,B 0,C 180,E1 -17580.479,E2 -17580.479} C_VEL
LIN {X 0,Y 277.265,Z 194.875,A -85,B 0,C 180,E1 -17583.889,E2 -17583.889} C_VEL
LIN {X 0,Y 277.235,Z 193.254,A -85,B 0,C 180,E1 -17585.785,E2 -17585.785} C_VEL
LIN {X 0,Y 277.245,Z 192.952,A -85,B 0,C 180,E1 -17588.201,E2 -17588.201} C_VEL
LIN {X 0,Y 277.222,Z 192.953,A -85,B 0,C 180,E1 -17592.676,E2 -17592.676} C_VEL
LIN {X 0,Y 277.25,Z 192.95,A -85,B 0,C 180,E1 -17596.809,E2 -17596.809} C_VEL
LIN {X 0,Y 277.252,Z 192.949,A -85,B 0,C 180,E1 -17600.674,E2 -17600.674} C_VEL
LIN {X 0,Y 277.272,Z 192.946,A -85,B 0,C 180,E1 -17604.339,E2 -17604.339} C_VEL
LIN {X 0,Y 277.226,Z 192.949,A -85,B 0,C 180,E1 -17607.833,E2 -17607.833} C_VEL
LIN {X 0,Y 277.251,Z 192.948,A -85,B 0,C 180,E1 -17611.208,E2 -17611.208} C_VEL
LIN {X 0,Y 277.3,Z 192.943,A -85,B 0,C 180,E1 -17614.478,E2 -17614.478} C_VEL
LIN {X 0,Y 277.287,Z 192.93,A -85,B 0,C 180,E1 -17617.654,E2 -17617.654} C_VEL
LIN {X 0,Y 277.349,Z 192.922,A -85,B 0,C 180,E1 -17620.766,E2 -17620.766} C_VEL
LIN {X 0,Y 277.405,Z 192.928,A -85,B 0,C 180,E1 -17625.324,E2 -17625.324} C_VEL
LIN {X 0,Y 277.53,Z 192.908,A -85,B 0,C 180,E1 -17629.789,E2 -17629.789} C_VEL
LIN {X 0,Y 277.639,Z 192.899,A -85,B 0,C 180,E1 -17632.728,E2 -17632.728} C_VEL
LIN {X 0,Y 277.793,Z 192.879,A -85,B 0,C 180,E1 -17638.55,E2 -17638.55} C_VEL
LIN {X 0,Y 277.799,Z 192.881,A -85,B 0,C 180,E1 -17641.449,E2 -17641.449} C_VEL
LIN {X 0,Y 277.549,Z 192.913,A -85,B 0,C 180,E1 -17645.813,E2 -17645.813} C_VEL
LIN {X 0,Y 277.606,Z 192.906,A -85,B 0,C 180,E1 -17649.158,E2 -17649.158} C_VEL
LIN {X 0,Y 277.409,Z 192.929,A -85,B 0,C 180,E1 -17651.45,E2 -17651.45} C_VEL
LIN {X 0,Y 276.728,Z 193.018,A -85,B 0,C 180,E1 -17652.663,E2 -17652.663} C_VEL
LIN {X 0,Y 273.821,Z 193.378,A -85,B 0,C 180,E1 -17654.636,E2 -17654.636} C_VEL
LIN {X 0,Y 271.369,Z 193.681,A -85,B 0,C 180,E1 -17656.24,E2 -17656.24} C_VEL
LIN {X 0,Y 270.338,Z 193.812,A -85,B 0,C 180,E1 -17657.485,E2 -17657.485} C_VEL
LIN {X 0,Y 270.265,Z 193.817,A -85,B 0,C 180,E1 -17657.907,E2 -17657.907} C_VEL
LIN {X 0,Y 270.243,Z 193.824,A -85,B 0,C 180,E1 -17661.351,E2 -17661.351} C_VEL
LIN {X 0,Y 270.258,Z 193.821,A -85,B 0,C 180,E1 -17664.587,E2 -17664.587} C_VEL
LIN {X 0,Y 270.252,Z 193.819,A -85,B 0,C 180,E1 -17667.911,E2 -17667.911} C_VEL
LIN {X 0,Y 270.165,Z 193.826,A -85,B 0,C 180,E1 -17671.35,E2 -17671.35} C_VEL
LIN {X 0,Y 270.197,Z 193.83,A -85,B 0,C 180,E1 -17674.906,E2 -17674.906} C_VEL
LIN {X 0,Y 270.207,Z 193.828,A -85,B 0,C 180,E1 -17678.72,E2 -17678.72} C_VEL
LIN {X 0,Y 270.278,Z 193.859,A -85,B 0,C 180,E1 -17682.926,E2 -17682.926} C_VEL
LIN {X 0,Y 270.895,Z 197.422,A -85,B 0,C 180,E1 -17686.587,E2 -17686.587} C_VEL
LIN {X 0,Y 271.575,Z 201.956,A -85,B 0,C 180,E1 -17690.928,E2 -17690.928} C_VEL
LIN {X 0,Y 271.757,Z 204.835,A -85,B 0,C 180,E1 -17693.505,E2 -17693.505} C_VEL
LIN {X 0,Y 271.483,Z 207.688,A -85,B 0,C 180,E1 -17695.934,E2 -17695.934} C_VEL
LIN {X 0,Y 270.883,Z 211.27,A -85,B 0,C 180,E1 -17698.89,E2 -17698.89} C_VEL
LIN {X 0,Y 269.952,Z 216.893,A -85,B 0,C 180,E1 -17703.422,E2 -17703.422} C_VEL
LIN {X 0,Y 273.353,Z 231.124,A -85,B 0,C 180,E1 -17704.489,E2 -17704.489} C_VEL
LIN {X 0,Y 275.468,Z 242.986,A -85,B 0,C 180,E1 -17705.58,E2 -17705.58} C_VEL
LIN {X 0,Y 276.71,Z 254.473,A -85,B 0,C 180,E1 -17706.835,E2 -17706.835} C_VEL
LIN {X 0,Y 277.323,Z 265.308,A -85,B 0,C 180,E1 -17708.248,E2 -17708.248} C_VEL
LIN {X 0,Y 275.456,Z 276.356,A -85,B 0,C 180,E1 -17709.855,E2 -17709.855} C_VEL
LIN {X 0,Y 273.665,Z 286.406,A -85,B 0,C 180,E1 -17711.705,E2 -17711.705} C_VEL
LIN {X 0,Y 272.28,Z 294.321,A -85,B 0,C 180,E1 -17713.507,E2 -17713.507} C_VEL
LIN {X 0,Y 270.787,Z 302.262,A -85,B 0,C 180,E1 -17715.728,E2 -17715.728} C_VEL
LIN {X 0,Y 269.619,Z 308.602,A -85,B 0,C 180,E1 -17717.966,E2 -17717.966} C_VEL
LIN {X 0,Y 268.912,Z 313.652,A -85,B 0,C 180,E1 -17720.221,E2 -17720.221} C_VEL
LIN {X 0,Y 268.426,Z 317.562,A -85,B 0,C 180,E1 -17722.479,E2 -17722.479} C_VEL
LIN {X 0,Y 268.171,Z 320.493,A -85,B 0,C 180,E1 -17724.793,E2 -17724.793} C_VEL
LIN {X 0,Y 268.167,Z 322.36,A -85,B 0,C 180,E1 -17726.997,E2 -17726.997} C_VEL
LIN {X 0,Y 268.188,Z 323.103,A -85,B 0,C 180,E1 -17728.499,E2 -17728.499} C_VEL
LIN {X 0,Y 268.2,Z 323.453,A -85,B 0,C 180,E1 -17730.001,E2 -17730.001} C_VEL
LIN {X 0,Y 268.181,Z 323.416,A -85,B 0,C 180,E1 -17731.503,E2 -17731.503} C_VEL
LIN {X 0,Y 268.155,Z 322.989,A -85,B 0,C 180,E1 -17733.005,E2 -17733.005} C_VEL
LIN {X 0,Y 268.163,Z 321.613,A -85,B 0,C 180,E1 -17735.188,E2 -17735.188} C_VEL
LIN {X 0,Y 268.563,Z 318.19,A -85,B 0,C 180,E1 -17738.276,E2 -17738.276} C_VEL
LIN {X 0,Y 269.208,Z 314.507,A -85,B 0,C 180,E1 -17740.53,E2 -17740.53} C_VEL
LIN {X 0,Y 270.082,Z 309.714,A -85,B 0,C 180,E1 -17742.779,E2 -17742.779} C_VEL
LIN {X 0,Y 271.748,Z 302.555,A -85,B 0,C 180,E1 -17745.372,E2 -17745.372} C_VEL
LIN {X 0,Y 273.444,Z 294.746,A -85,B 0,C 180,E1 -17747.577,E2 -17747.577} C_VEL
LIN {X 0,Y 275.059,Z 286.783,A -85,B 0,C 180,E1 -17749.4,E2 -17749.4} C_VEL
LIN {X 0,Y 277.053,Z 277.079,A -85,B 0,C 180,E1 -17751.19,E2 -17751.19} C_VEL
LIN {X 0,Y 278.926,Z 267.596,A -85,B 0,C 180,E1 -17752.596,E2 -17752.596} C_VEL
LIN {X 0,Y 278.503,Z 257.681,A -85,B 0,C 180,E1 -17753.979,E2 -17753.979} C_VEL
LIN {X 0,Y 277.207,Z 246.344,A -85,B 0,C 180,E1 -17755.348,E2 -17755.348} C_VEL
LIN {X 0,Y 275.046,Z 234.4,A -85,B 0,C 180,E1 -17756.579,E2 -17756.579} C_VEL
LIN {X 0,Y 271.665,Z 221.623,A -85,B 0,C 180,E1 -17757.71,E2 -17757.71} C_VEL
LIN {X 0,Y 270.41,Z 216.73,A -85,B 0,C 180,E1 -17758.082,E2 -17758.082} C_VEL
LIN {X 0,Y 271.101,Z 212.845,A -85,B 0,C 180,E1 -17761.229,E2 -17761.229} C_VEL
LIN {X 0,Y 271.821,Z 208.774,A -85,B 0,C 180,E1 -17764.666,E2 -17764.666} C_VEL
LIN {X 0,Y 271.962,Z 206.402,A -85,B 0,C 180,E1 -17766.765,E2 -17766.765} C_VEL
LIN {X 0,Y 271.846,Z 203.811,A -85,B 0,C 180,E1 -17769.142,E2 -17769.142} C_VEL
LIN {X 0,Y 271.433,Z 200.555,A -85,B 0,C 180,E1 -17772.312,E2 -17772.312} C_VEL
LIN {X 0,Y 270.659,Z 196.422,A -85,B 0,C 180,E1 -17776.637,E2 -17776.637} C_VEL
LIN {X 0,Y 270.204,Z 193.829,A -85,B 0,C 180,E1 -17779.685,E2 -17779.685} C_VEL
LIN {X 0,Y 270.215,Z 193.829,A -85,B 0,C 180,E1 -17783.73,E2 -17783.73} C_VEL
LIN {X 0,Y 270.19,Z 193.832,A -85,B 0,C 180,E1 -17786.891,E2 -17786.891} C_VEL
LIN {X 0,Y 270.181,Z 193.831,A -85,B 0,C 180,E1 -17790.381,E2 -17790.381} C_VEL
LIN {X 0,Y 270.25,Z 193.821,A -85,B 0,C 180,E1 -17793.763,E2 -17793.763} C_VEL
LIN {X 0,Y 270.24,Z 193.824,A -85,B 0,C 180,E1 -17797.04,E2 -17797.04} C_VEL
LIN {X 0,Y 270.314,Z 193.813,A -85,B 0,C 180,E1 -17800.246,E2 -17800.246} C_VEL
LIN {X 0,Y 270.381,Z 193.806,A -85,B 0,C 180,E1 -17804.934,E2 -17804.934} C_VEL
LIN {X 0,Y 270.398,Z 193.801,A -85,B 0,C 180,E1 -17809.518,E2 -17809.518} C_VEL
LIN {X 0,Y 270.585,Z 193.78,A -85,B 0,C 180,E1 -17812.538,E2 -17812.538} C_VEL
LIN {X 0,Y 270.767,Z 193.758,A -85,B 0,C 180,E1 -17818.513,E2 -17818.513} C_VEL
LIN {X 0,Y 270.775,Z 193.754,A -85,B 0,C 180,E1 -17821.488,E2 -17821.488} C_VEL
LIN {X 0,Y 270.528,Z 193.784,A -85,B 0,C 180,E1 -17826.71,E2 -17826.71} C_VEL
LIN {X 0,Y 270.511,Z 193.787,A -85,B 0,C 180,E1 -17829.176,E2 -17829.176} C_VEL
LIN {X 0,Y 270.34,Z 193.811,A -85,B 0,C 180,E1 -17833.531,E2 -17833.531} C_VEL
LIN {X 0,Y 270.32,Z 193.811,A -85,B 0,C 180,E1 -17836.618,E2 -17836.618} C_VEL
LIN {X 0,Y 270.28,Z 193.816,A -85,B 0,C 180,E1 -17840.602,E2 -17840.602} C_VEL
LIN {X 0,Y 270.262,Z 193.818,A -85,B 0,C 180,E1 -17844.587,E2 -17844.587} C_VEL
LIN {X 0,Y 270.26,Z 193.819,A -85,B 0,C 180,E1 -17847.91,E2 -17847.91} C_VEL
LIN {X 0,Y 270.175,Z 193.832,A -85,B 0,C 180,E1 -17851.35,E2 -17851.35} C_VEL
LIN {X 0,Y 270.192,Z 193.831,A -85,B 0,C 180,E1 -17854.908,E2 -17854.908} C_VEL
LIN {X 0,Y 270.191,Z 193.83,A -85,B 0,C 180,E1 -17858.712,E2 -17858.712} C_VEL
LIN {X 0,Y 270.159,Z 193.833,A -85,B 0,C 180,E1 -17863.251,E2 -17863.251} C_VEL
LIN {X 0,Y 270.174,Z 193.928,A -85,B 0,C 180,E1 -17867.445,E2 -17867.445} C_VEL
LIN {X 0,Y 270.455,Z 196.866,A -85,B 0,C 180,E1 -17871.223,E2 -17871.223} C_VEL
LIN {X 0,Y 270.42,Z 198.87,A -85,B 0,C 180,E1 -17873.676,E2 -17873.676} C_VEL
LIN {X 0,Y 270.094,Z 201.674,A -85,B 0,C 180,E1 -17876.879,E2 -17876.879} C_VEL
LIN {X 0,Y 269.812,Z 204.364,A -85,B 0,C 180,E1 -17879.906,E2 -17879.906} C_VEL
LIN {X 0,Y 274.79,Z 219.312,A -85,B 0,C 180,E1 -17881.335,E2 -17881.335} C_VEL
LIN {X 0,Y 277.736,Z 230.535,A -85,B 0,C 180,E1 -17882.567,E2 -17882.567} C_VEL
LIN {X 0,Y 279.654,Z 240.72,A -85,B 0,C 180,E1 -17883.831,E2 -17883.831} C_VEL
LIN {X 0,Y 280.648,Z 249.183,A -85,B 0,C 180,E1 -17885.009,E2 -17885.009} C_VEL
LIN {X 0,Y 278.618,Z 260.564,A -85,B 0,C 180,E1 -17886.592,E2 -17886.592} C_VEL
LIN {X 0,Y 276.555,Z 270.626,A -85,B 0,C 180,E1 -17888.378,E2 -17888.378} C_VEL
LIN {X 0,Y 274.752,Z 278.845,A -85,B 0,C 180,E1 -17890.189,E2 -17890.189} C_VEL
LIN {X 0,Y 272.914,Z 286.708,A -85,B 0,C 180,E1 -17892.331,E2 -17892.331} C_VEL
LIN {X 0,Y 271.794,Z 292.334,A -85,B 0,C 180,E1 -17894.246,E2 -17894.246} C_VEL
LIN {X 0,Y 270.397,Z 297.66,A -85,B 0,C 180,E1 -17896.472,E2 -17896.472} C_VEL
LIN {X 0,Y 269.513,Z 301.806,A -85,B 0,C 180,E1 -17898.721,E2 -17898.721} C_VEL
LIN {X 0,Y 268.876,Z 304.897,A -85,B 0,C 180,E1 -17900.977,E2 -17900.977} C_VEL
LIN {X 0,Y 268.553,Z 306.434,A -85,B 0,C 180,E1 -17902.481,E2 -17902.481} C_VEL
LIN {X 0,Y 268.36,Z 307.735,A -85,B 0,C 180,E1 -17904.374,E2 -17904.374} C_VEL
LIN {X 0,Y 268.252,Z 308.53,A -85,B 0,C 180,E1 -17906.996,E2 -17906.996} C_VEL
LIN {X 0,Y 268.217,Z 308.462,A -85,B 0,C 180,E1 -17908.498,E2 -17908.498} C_VEL
LIN {X 0,Y 268.21,Z 307.988,A -85,B 0,C 180,E1 -17909.999,E2 -17909.999} C_VEL
LIN {X 0,Y 268.496,Z 305.823,A -85,B 0,C 180,E1 -17913,E2 -17913} C_VEL
LIN {X 0,Y 268.961,Z 303.122,A -85,B 0,C 180,E1 -17915.246,E2 -17915.246} C_VEL
LIN {X 0,Y 269.673,Z 298.51,A -85,B 0,C 180,E1 -17917.971,E2 -17917.971} C_VEL
LIN {X 0,Y 270.674,Z 292.743,A -85,B 0,C 180,E1 -17920.47,E2 -17920.47} C_VEL
LIN {X 0,Y 271.899,Z 286.194,A -85,B 0,C 180,E1 -17922.69,E2 -17922.69} C_VEL
LIN {X 0,Y 273.61,Z 278.051,A -85,B 0,C 180,E1 -17924.882,E2 -17924.882} C_VEL
LIN {X 0,Y 275.154,Z 269.726,A -85,B 0,C 180,E1 -17926.697,E2 -17926.697} C_VEL
LIN {X 0,Y 276.843,Z 259.462,A -85,B 0,C 180,E1 -17928.499,E2 -17928.499} C_VEL
LIN {X 0,Y 278.241,Z 251.207,A -85,B 0,C 180,E1 -17929.675,E2 -17929.675} C_VEL
LIN {X 0,Y 278.885,Z 245.408,A -85,B 0,C 180,E1 -17930.397,E2 -17930.397} C_VEL
LIN {X 0,Y 277.512,Z 235.056,A -85,B 0,C 180,E1 -17931.694,E2 -17931.694} C_VEL
LIN {X 0,Y 274.904,Z 222.766,A -85,B 0,C 180,E1 -17933.021,E2 -17933.021} C_VEL
LIN {X 0,Y 271.395,Z 210.168,A -85,B 0,C 180,E1 -17934.163,E2 -17934.163} C_VEL
LIN {X 0,Y 269.493,Z 204.217,A -85,B 0,C 180,E1 -17934.659,E2 -17934.659} C_VEL
LIN {X 0,Y 269.829,Z 201.165,A -85,B 0,C 180,E1 -17937.955,E2 -17937.955} C_VEL
LIN {X 0,Y 270.111,Z 198.138,A -85,B 0,C 180,E1 -17941.354,E2 -17941.354} C_VEL
LIN {X 0,Y 270.222,Z 195.089,A -85,B 0,C 180,E1 -17944.898,E2 -17944.898} C_VEL
LIN {X 0,Y 270.15,Z 193.839,A -85,B 0,C 180,E1 -17946.747,E2 -17946.747} C_VEL
LIN {X 0,Y 270.167,Z 193.832,A -85,B 0,C 180,E1 -17950.562,E2 -17950.562} C_VEL
LIN {X 0,Y 270.177,Z 193.831,A -85,B 0,C 180,E1 -17954.609,E2 -17954.609} C_VEL
LIN {X 0,Y 270.253,Z 193.823,A -85,B 0,C 180,E1 -17958.945,E2 -17958.945} C_VEL
LIN {X 0,Y 270.219,Z 193.826,A -85,B 0,C 180,E1 -17963.258,E2 -17963.258} C_VEL
LIN {X 0,Y 270.185,Z 193.83,A -85,B 0,C 180,E1 -17966.889,E2 -17966.889} C_VEL
LIN {X 0,Y 270.178,Z 193.831,A -85,B 0,C 180,E1 -17970.38,E2 -17970.38} C_VEL
LIN {X 0,Y 270.247,Z 193.82,A -85,B 0,C 180,E1 -17973.762,E2 -17973.762} C_VEL
LIN {X 0,Y 270.232,Z 193.809,A -85,B 0,C 180,E1 -17977.038,E2 -17977.038} C_VEL
LIN {X 0,Y 270.306,Z 193.792,A -85,B 0,C 180,E1 -17980.244,E2 -17980.244} C_VEL
LIN {X 0,Y 270.374,Z 193.804,A -85,B 0,C 180,E1 -17984.933,E2 -17984.933} C_VEL
LIN {X 0,Y 270.472,Z 193.786,A -85,B 0,C 180,E1 -17989.52,E2 -17989.52} C_VEL
LIN {X 0,Y 270.597,Z 193.777,A -85,B 0,C 180,E1 -17992.538,E2 -17992.538} C_VEL
LIN {X 0,Y 270.759,Z 193.756,A -85,B 0,C 180,E1 -17998.512,E2 -17998.512} C_VEL
LIN {X 0,Y 270.766,Z 193.758,A -85,B 0,C 180,E1 -18001.487,E2 -18001.487} C_VEL
LIN {X 0,Y 270.585,Z 193.781,A -85,B 0,C 180,E1 -18007.462,E2 -18007.462} C_VEL
LIN {X 0,Y 270.418,Z 193.799,A -85,B 0,C 180,E1 -18010.482,E2 -18010.482} C_VEL
LIN {X 0,Y 270.359,Z 193.809,A -85,B 0,C 180,E1 -18015.067,E2 -18015.067} C_VEL
LIN {X 0,Y 270.265,Z 193.817,A -85,B 0,C 180,E1 -18017.907,E2 -18017.907} C_VEL
LIN {X 0,Y 269.61,Z 193.903,A -85,B 0,C 180,E1 -18019.151,E2 -18019.151} C_VEL
LIN {X 0,Y 266.715,Z 194.264,A -85,B 0,C 180,E1 -18021.176,E2 -18021.176} C_VEL
LIN {X 0,Y 264.268,Z 194.569,A -85,B 0,C 180,E1 -18022.823,E2 -18022.823} C_VEL
LIN {X 0,Y 263.254,Z 194.692,A -85,B 0,C 180,E1 -18024.102,E2 -18024.102} C_VEL
LIN {X 0,Y 263.192,Z 194.7,A -85,B 0,C 180,E1 -18024.535,E2 -18024.535} C_VEL
LIN {X 0,Y 263.16,Z 194.703,A -85,B 0,C 180,E1 -18028.732,E2 -18028.732} C_VEL
LIN {X 0,Y 263.115,Z 194.706,A -85,B 0,C 180,E1 -18032.291,E2 -18032.291} C_VEL
LIN {X 0,Y 263.17,Z 194.703,A -85,B 0,C 180,E1 -18035.981,E2 -18035.981} C_VEL
LIN {X 0,Y 263.145,Z 194.707,A -85,B 0,C 180,E1 -18039.865,E2 -18039.865} C_VEL
LIN {X 0,Y 263.271,Z 194.909,A -85,B 0,C 180,E1 -18042.639,E2 -18042.639} C_VEL
LIN {X 0,Y 263.852,Z 198.225,A -85,B 0,C 180,E1 -18046.174,E2 -18046.174} C_VEL
LIN {X 0,Y 264.469,Z 202.514,A -85,B 0,C 180,E1 -18050.412,E2 -18050.412} C_VEL
LIN {X 0,Y 264.719,Z 205.054,A -85,B 0,C 180,E1 -18052.794,E2 -18052.794} C_VEL
LIN {X 0,Y 264.551,Z 208.043,A -85,B 0,C 180,E1 -18055.441,E2 -18055.441} C_VEL
LIN {X 0,Y 263.631,Z 212.926,A -85,B 0,C 180,E1 -18059.572,E2 -18059.572} C_VEL
LIN {X 0,Y 263.001,Z 216.738,A -85,B 0,C 180,E1 -18062.708,E2 -18062.708} C_VEL
LIN {X 0,Y 266.272,Z 230.077,A -85,B 0,C 180,E1 -18063.732,E2 -18063.732} C_VEL
LIN {X 0,Y 268.271,Z 240.397,A -85,B 0,C 180,E1 -18064.695,E2 -18064.695} C_VEL
LIN {X 0,Y 269.776,Z 252.783,A -85,B 0,C 180,E1 -18066.061,E2 -18066.061} C_VEL
LIN {X 0,Y 270.522,Z 264.919,A -85,B 0,C 180,E1 -18067.672,E2 -18067.672} C_VEL
LIN {X 0,Y 269.205,Z 273.762,A -85,B 0,C 180,E1 -18068.966,E2 -18068.966} C_VEL
LIN {X 0,Y 267.269,Z 284.123,A -85,B 0,C 180,E1 -18070.813,E2 -18070.813} C_VEL
LIN {X 0,Y 265.74,Z 292.818,A -85,B 0,C 180,E1 -18072.768,E2 -18072.768} C_VEL
LIN {X 0,Y 264.151,Z 300.757,A -85,B 0,C 180,E1 -18074.967,E2 -18074.967} C_VEL
LIN {X 0,Y 263.004,Z 306.36,A -85,B 0,C 180,E1 -18076.873,E2 -18076.873} C_VEL
LIN {X 0,Y 262.081,Z 311.84,A -85,B 0,C 180,E1 -18079.183,E2 -18079.183} C_VEL
LIN {X 0,Y 261.507,Z 316.13,A -85,B 0,C 180,E1 -18081.501,E2 -18081.501} C_VEL
LIN {X 0,Y 261.155,Z 319.349,A -85,B 0,C 180,E1 -18083.822,E2 -18083.822} C_VEL
LIN {X 0,Y 261.066,Z 320.953,A -85,B 0,C 180,E1 -18085.369,E2 -18085.369} C_VEL
LIN {X 0,Y 261.063,Z 322.148,A -85,B 0,C 180,E1 -18086.915,E2 -18086.915} C_VEL
LIN {X 0,Y 261.115,Z 322.898,A -85,B 0,C 180,E1 -18088.459,E2 -18088.459} C_VEL
LIN {X 0,Y 261.126,Z 323.254,A -85,B 0,C 180,E1 -18090.001,E2 -18090.001} C_VEL
LIN {X 0,Y 261.108,Z 323.221,A -85,B 0,C 180,E1 -18091.543,E2 -18091.543} C_VEL
LIN {X 0,Y 261.05,Z 322.8,A -85,B 0,C 180,E1 -18093.087,E2 -18093.087} C_VEL
LIN {X 0,Y 261.085,Z 321.574,A -85,B 0,C 180,E1 -18095.138,E2 -18095.138} C_VEL
LIN {X 0,Y 261.356,Z 319.025,A -85,B 0,C 180,E1 -18097.727,E2 -18097.727} C_VEL
LIN {X 0,Y 261.948,Z 315.695,A -85,B 0,C 180,E1 -18100.044,E2 -18100.044} C_VEL
LIN {X 0,Y 262.765,Z 311.297,A -85,B 0,C 180,E1 -18102.355,E2 -18102.355} C_VEL
LIN {X 0,Y 264.075,Z 305.716,A -85,B 0,C 180,E1 -18104.645,E2 -18104.645} C_VEL
LIN {X 0,Y 265.683,Z 298.756,A -85,B 0,C 180,E1 -18106.916,E2 -18106.916} C_VEL
LIN {X 0,Y 267.574,Z 290.194,A -85,B 0,C 180,E1 -18109.129,E2 -18109.129} C_VEL
LIN {X 0,Y 269.584,Z 281.128,A -85,B 0,C 180,E1 -18111.005,E2 -18111.005} C_VEL
LIN {X 0,Y 271.686,Z 271.342,A -85,B 0,C 180,E1 -18112.63,E2 -18112.63} C_VEL
LIN {X 0,Y 272.259,Z 267.559,A -85,B 0,C 180,E1 -18113.182,E2 -18113.182} C_VEL
LIN {X 0,Y 271.723,Z 256.798,A -85,B 0,C 180,E1 -18114.731,E2 -18114.731} C_VEL
LIN {X 0,Y 270.431,Z 245.869,A -85,B 0,C 180,E1 -18116.085,E2 -18116.085} C_VEL
LIN {X 0,Y 268.155,Z 233.941,A -85,B 0,C 180,E1 -18117.364,E2 -18117.364} C_VEL
LIN {X 0,Y 264.752,Z 221.139,A -85,B 0,C 180,E1 -18118.542,E2 -18118.542} C_VEL
LIN {X 0,Y 263.532,Z 216.517,A -85,B 0,C 180,E1 -18118.907,E2 -18118.907} C_VEL
LIN {X 0,Y 264.43,Z 211.683,A -85,B 0,C 180,E1 -18123.013,E2 -18123.013} C_VEL
LIN {X 0,Y 264.888,Z 208.616,A -85,B 0,C 180,E1 -18125.71,E2 -18125.71} C_VEL
LIN {X 0,Y 264.89,Z 205.536,A -85,B 0,C 180,E1 -18128.57,E2 -18128.57} C_VEL
LIN {X 0,Y 264.494,Z 202.16,A -85,B 0,C 180,E1 -18131.927,E2 -18131.927} C_VEL
LIN {X 0,Y 263.774,Z 198.195,A -85,B 0,C 180,E1 -18136.152,E2 -18136.152} C_VEL
LIN {X 0,Y 263.132,Z 194.709,A -85,B 0,C 180,E1 -18140.322,E2 -18140.322} C_VEL
LIN {X 0,Y 263.153,Z 194.709,A -85,B 0,C 180,E1 -18144.017,E2 -18144.017} C_VEL
LIN {X 0,Y 263.117,Z 194.714,A -85,B 0,C 180,E1 -18147.71,E2 -18147.71} C_VEL
LIN {X 0,Y 263.168,Z 194.704,A -85,B 0,C 180,E1 -18151.791,E2 -18151.791} C_VEL
LIN {X 0,Y 263.217,Z 194.698,A -85,B 0,C 180,E1 -18155.198,E2 -18155.198} C_VEL
LIN {X 0,Y 263.276,Z 194.689,A -85,B 0,C 180,E1 -18159.695,E2 -18159.695} C_VEL
LIN {X 0,Y 263.33,Z 194.685,A -85,B 0,C 180,E1 -18164.521,E2 -18164.521} C_VEL
LIN {X 0,Y 263.34,Z 194.681,A -85,B 0,C 180,E1 -18169.233,E2 -18169.233} C_VEL
LIN {X 0,Y 263.545,Z 194.658,A -85,B 0,C 180,E1 -18172.338,E2 -18172.338} C_VEL
LIN {X 0,Y 263.732,Z 194.635,A -85,B 0,C 180,E1 -18178.473,E2 -18178.473} C_VEL
LIN {X 0,Y 263.741,Z 194.631,A -85,B 0,C 180,E1 -18181.527,E2 -18181.527} C_VEL
LIN {X 0,Y 263.54,Z 194.657,A -85,B 0,C 180,E1 -18187.663,E2 -18187.663} C_VEL
LIN {X 0,Y 263.305,Z 194.686,A -85,B 0,C 180,E1 -18192.33,E2 -18192.33} C_VEL
LIN {X 0,Y 263.308,Z 194.686,A -85,B 0,C 180,E1 -18196.089,E2 -18196.089} C_VEL
LIN {X 0,Y 263.251,Z 194.692,A -85,B 0,C 180,E1 -18200.308,E2 -18200.308} C_VEL
LIN {X 0,Y 263.197,Z 194.701,A -85,B 0,C 180,E1 -18205.293,E2 -18205.293} C_VEL
LIN {X 0,Y 263.156,Z 194.704,A -85,B 0,C 180,E1 -18208.733,E2 -18208.733} C_VEL
LIN {X 0,Y 263.124,Z 194.708,A -85,B 0,C 180,E1 -18212.29,E2 -18212.29} C_VEL
LIN {X 0,Y 263.173,Z 194.704,A -85,B 0,C 180,E1 -18216.764,E2 -18216.764} C_VEL
LIN {X 0,Y 263.099,Z 194.71,A -85,B 0,C 180,E1 -18219.874,E2 -18219.874} C_VEL
LIN {X 0,Y 263.098,Z 194.712,A -85,B 0,C 180,E1 -18223.99,E2 -18223.99} C_VEL
LIN {X 0,Y 263.078,Z 194.716,A -85,B 0,C 180,E1 -18226.162,E2 -18226.162} C_VEL
LIN {X 0,Y 263.237,Z 195.82,A -85,B 0,C 180,E1 -18228.38,E2 -18228.38} C_VEL
LIN {X 0,Y 263.413,Z 198.743,A -85,B 0,C 180,E1 -18232.148,E2 -18232.148} C_VEL
LIN {X 0,Y 263.35,Z 200.272,A -85,B 0,C 180,E1 -18234.049,E2 -18234.049} C_VEL
LIN {X 0,Y 262.934,Z 203.381,A -85,B 0,C 180,E1 -18237.686,E2 -18237.686} C_VEL
LIN {X 0,Y 262.854,Z 204.592,A -85,B 0,C 180,E1 -18239.066,E2 -18239.066} C_VEL
LIN {X 0,Y 264.872,Z 210.471,A -85,B 0,C 180,E1 -18239.621,E2 -18239.621} C_VEL
LIN {X 0,Y 268.662,Z 222.013,A -85,B 0,C 180,E1 -18240.832,E2 -18240.832} C_VEL
LIN {X 0,Y 271.611,Z 233.894,A -85,B 0,C 180,E1 -18242.242,E2 -18242.242} C_VEL
LIN {X 0,Y 273.339,Z 244.095,A -85,B 0,C 180,E1 -18243.606,E2 -18243.606} C_VEL
LIN {X 0,Y 274.024,Z 250.292,A -85,B 0,C 180,E1 -18244.522,E2 -18244.522} C_VEL
LIN {X 0,Y 272.108,Z 260.587,A -85,B 0,C 180,E1 -18245.997,E2 -18245.997} C_VEL
LIN {X 0,Y 269.949,Z 270.69,A -85,B 0,C 180,E1 -18247.822,E2 -18247.822} C_VEL
LIN {X 0,Y 268.055,Z 278.931,A -85,B 0,C 180,E1 -18249.672,E2 -18249.672} C_VEL
LIN {X 0,Y 266.017,Z 287.284,A -85,B 0,C 180,E1 -18252.01,E2 -18252.01} C_VEL
LIN {X 0,Y 264.452,Z 294.382,A -85,B 0,C 180,E1 -18254.588,E2 -18254.588} C_VEL
LIN {X 0,Y 263.092,Z 299.309,A -85,B 0,C 180,E1 -18256.876,E2 -18256.876} C_VEL
LIN {X 0,Y 262.278,Z 303.107,A -85,B 0,C 180,E1 -18259.189,E2 -18259.189} C_VEL
LIN {X 0,Y 261.85,Z 305.061,A -85,B 0,C 180,E1 -18260.732,E2 -18260.732} C_VEL
LIN {X 0,Y 261.511,Z 306.604,A -85,B 0,C 180,E1 -18262.277,E2 -18262.277} C_VEL
LIN {X 0,Y 261.282,Z 308.014,A -85,B 0,C 180,E1 -18264.41,E2 -18264.41} C_VEL
LIN {X 0,Y 261.165,Z 308.724,A -85,B 0,C 180,E1 -18266.914,E2 -18266.914} C_VEL
LIN {X 0,Y 261.145,Z 308.662,A -85,B 0,C 180,E1 -18268.457,E2 -18268.457} C_VEL
LIN {X 0,Y 261.136,Z 308.2,A -85,B 0,C 180,E1 -18269.999,E2 -18269.999} C_VEL
LIN {X 0,Y 261.434,Z 306.047,A -85,B 0,C 180,E1 -18273.081,E2 -18273.081} C_VEL
LIN {X 0,Y 261.901,Z 303.359,A -85,B 0,C 180,E1 -18275.388,E2 -18275.388} C_VEL
LIN {X 0,Y 262.558,Z 299.211,A -85,B 0,C 180,E1 -18277.942,E2 -18277.942} C_VEL
LIN {X 0,Y 263.346,Z 294.874,A -85,B 0,C 180,E1 -18279.988,E2 -18279.988} C_VEL
LIN {X 0,Y 264.504,Z 288.822,A -85,B 0,C 180,E1 -18282.271,E2 -18282.271} C_VEL
LIN {X 0,Y 266.189,Z 281.291,A -85,B 0,C 180,E1 -18284.524,E2 -18284.524} C_VEL
LIN {X 0,Y 267.697,Z 273.59,A -85,B 0,C 180,E1 -18286.391,E2 -18286.391} C_VEL
LIN {X 0,Y 269.578,Z 263.126,A -85,B 0,C 180,E1 -18288.425,E2 -18288.425} C_VEL
LIN {X 0,Y 271.093,Z 253.97,A -85,B 0,C 180,E1 -18289.857,E2 -18289.857} C_VEL
LIN {X 0,Y 272.099,Z 248.296,A -85,B 0,C 180,E1 -18290.6,E2 -18290.6} C_VEL
LIN {X 0,Y 271.87,Z 243.765,A -85,B 0,C 180,E1 -18291.215,E2 -18291.215} C_VEL
LIN {X 0,Y 270.219,Z 232.944,A -85,B 0,C 180,E1 -18292.584,E2 -18292.584} C_VEL
LIN {X 0,Y 267.716,Z 221.66,A -85,B 0,C 180,E1 -18293.816,E2 -18293.816} C_VEL
LIN {X 0,Y 264.188,Z 209.836,A -85,B 0,C 180,E1 -18294.928,E2 -18294.928} C_VEL
LIN {X 0,Y 262.493,Z 204.448,A -85,B 0,C 180,E1 -18295.362,E2 -18295.362} C_VEL
LIN {X 0,Y 262.839,Z 201.399,A -85,B 0,C 180,E1 -18298.767,E2 -18298.767} C_VEL
LIN {X 0,Y 263.118,Z 198.35,A -85,B 0,C 180,E1 -18302.286,E2 -18302.286} C_VEL
LIN {X 0,Y 263.217,Z 196.793,A -85,B 0,C 180,E1 -18304.135,E2 -18304.135} C_VEL
LIN {X 0,Y 263.108,Z 194.717,A -85,B 0,C 180,E1 -18306.74,E2 -18306.74} C_VEL
LIN {X 0,Y 263.098,Z 194.714,A -85,B 0,C 180,E1 -18309.869,E2 -18309.869} C_VEL
LIN {X 0,Y 263.128,Z 194.709,A -85,B 0,C 180,E1 -18313.978,E2 -18313.978} C_VEL
LIN {X 0,Y 263.197,Z 194.699,A -85,B 0,C 180,E1 -18318.382,E2 -18318.382} C_VEL
LIN {X 0,Y 263.183,Z 194.703,A -85,B 0,C 180,E1 -18323.229,E2 -18323.229} C_VEL
LIN {X 0,Y 263.116,Z 194.707,A -85,B 0,C 180,E1 -18327.709,E2 -18327.709} C_VEL
LIN {X 0,Y 263.178,Z 194.7,A -85,B 0,C 180,E1 -18331.783,E2 -18331.783} C_VEL
LIN {X 0,Y 263.21,Z 194.692,A -85,B 0,C 180,E1 -18335.197,E2 -18335.197} C_VEL
LIN {X 0,Y 263.269,Z 194.664,A -85,B 0,C 180,E1 -18339.693,E2 -18339.693} C_VEL
LIN {X 0,Y 263.322,Z 194.685,A -85,B 0,C 180,E1 -18344.52,E2 -18344.52} C_VEL
LIN {X 0,Y 263.396,Z 194.666,A -85,B 0,C 180,E1 -18349.235,E2 -18349.235} C_VEL
LIN {X 0,Y 263.561,Z 194.655,A -85,B 0,C 180,E1 -18352.338,E2 -18352.338} C_VEL
LIN {X 0,Y 263.724,Z 194.632,A -85,B 0,C 180,E1 -18358.473,E2 -18358.473} C_VEL
LIN {X 0,Y 263.732,Z 194.634,A -85,B 0,C 180,E1 -18361.527,E2 -18361.527} C_VEL
LIN {X 0,Y 263.547,Z 194.659,A -85,B 0,C 180,E1 -18367.662,E2 -18367.662} C_VEL
LIN {X 0,Y 263.35,Z 194.681,A -85,B 0,C 180,E1 -18370.766,E2 -18370.766} C_VEL
LIN {X 0,Y 263.306,Z 194.688,A -85,B 0,C 180,E1 -18375.48,E2 -18375.48} C_VEL
LIN {X 0,Y 263.267,Z 194.691,A -85,B 0,C 180,E1 -18380.306,E2 -18380.306} C_VEL
LIN {X 0,Y 263.192,Z 194.7,A -85,B 0,C 180,E1 -18384.535,E2 -18384.535} C_VEL
LIN {X 0,Y 262.907,Z 194.739,A -85,B 0,C 180,E1 -18385.389,E2 -18385.389} C_VEL
LIN {X 0,Y 261.556,Z 194.907,A -85,B 0,C 180,E1 -18386.65,E2 -18386.65} C_VEL
LIN {X 0,Y 257.161,Z 195.444,A -85,B 0,C 180,E1 -18389.584,E2 -18389.584} C_VEL
LIN {X 0,Y 256.132,Z 195.57,A -85,B 0,C 180,E1 -18390.899,E2 -18390.899} C_VEL
LIN {X 0,Y 256.069,Z 195.58,A -85,B 0,C 180,E1 -18391.345,E2 -18391.345} C_VEL
LIN {X 0,Y 256.104,Z 195.584,A -85,B 0,C 180,E1 -18395.189,E2 -18395.189} C_VEL
LIN {X 0,Y 256.093,Z 195.585,A -85,B 0,C 180,E1 -18399.138,E2 -18399.138} C_VEL
LIN {X 0,Y 256.21,Z 195.728,A -85,B 0,C 180,E1 -18402.075,E2 -18402.075} C_VEL
LIN {X 0,Y 256.69,Z 198.729,A -85,B 0,C 180,E1 -18405.386,E2 -18405.386} C_VEL
LIN {X 0,Y 257.378,Z 203.076,A -85,B 0,C 180,E1 -18409.869,E2 -18409.869} C_VEL
LIN {X 0,Y 257.674,Z 206.463,A -85,B 0,C 180,E1 -18413.131,E2 -18413.131} C_VEL
LIN {X 0,Y 257.373,Z 209.589,A -85,B 0,C 180,E1 -18415.963,E2 -18415.963} C_VEL
LIN {X 0,Y 256.572,Z 213.723,A -85,B 0,C 180,E1 -18419.556,E2 -18419.556} C_VEL
LIN {X 0,Y 256.1,Z 216.476,A -85,B 0,C 180,E1 -18421.916,E2 -18421.916} C_VEL
LIN {X 0,Y 259.711,Z 231.247,A -85,B 0,C 180,E1 -18423.14,E2 -18423.14} C_VEL
LIN {X 0,Y 261.768,Z 242.297,A -85,B 0,C 180,E1 -18424.243,E2 -18424.243} C_VEL
LIN {X 0,Y 263.078,Z 253.732,A -85,B 0,C 180,E1 -18425.575,E2 -18425.575} C_VEL
LIN {X 0,Y 263.689,Z 264.526,A -85,B 0,C 180,E1 -18427.061,E2 -18427.061} C_VEL
LIN {X 0,Y 263.457,Z 268.541,A -85,B 0,C 180,E1 -18427.661,E2 -18427.661} C_VEL
LIN {X 0,Y 261.485,Z 278.911,A -85,B 0,C 180,E1 -18429.346,E2 -18429.346} C_VEL
LIN {X 0,Y 259.579,Z 288.721,A -85,B 0,C 180,E1 -18431.372,E2 -18431.372} C_VEL
LIN {X 0,Y 258.012,Z 296.581,A -85,B 0,C 180,E1 -18433.383,E2 -18433.383} C_VEL
LIN {X 0,Y 256.51,Z 303.979,A -85,B 0,C 180,E1 -18435.727,E2 -18435.727} C_VEL
LIN {X 0,Y 255.378,Z 309.915,A -85,B 0,C 180,E1 -18438.091,E2 -18438.091} C_VEL
LIN {X 0,Y 254.632,Z 314.601,A -85,B 0,C 180,E1 -18440.469,E2 -18440.469} C_VEL
LIN {X 0,Y 254.172,Z 318.172,A -85,B 0,C 180,E1 -18442.854,E2 -18442.854} C_VEL
LIN {X 0,Y 253.973,Z 320.732,A -85,B 0,C 180,E1 -18445.239,E2 -18445.239} C_VEL
LIN {X 0,Y 253.962,Z 321.934,A -85,B 0,C 180,E1 -18446.829,E2 -18446.829} C_VEL
LIN {X 0,Y 254.02,Z 322.693,A -85,B 0,C 180,E1 -18448.416,E2 -18448.416} C_VEL
LIN {X 0,Y 254.053,Z 323.054,A -85,B 0,C 180,E1 -18450.001,E2 -18450.001} C_VEL
LIN {X 0,Y 254.013,Z 323.026,A -85,B 0,C 180,E1 -18451.586,E2 -18451.586} C_VEL
LIN {X 0,Y 253.949,Z 322.61,A -85,B 0,C 180,E1 -18453.174,E2 -18453.174} C_VEL
LIN {X 0,Y 253.99,Z 321.566,A -85,B 0,C 180,E1 -18455.039,E2 -18455.039} C_VEL
LIN {X 0,Y 254.316,Z 318.855,A -85,B 0,C 180,E1 -18457.943,E2 -18457.943} C_VEL
LIN {X 0,Y 254.915,Z 315.535,A -85,B 0,C 180,E1 -18460.324,E2 -18460.324} C_VEL
LIN {X 0,Y 255.79,Z 311.149,A -85,B 0,C 180,E1 -18462.698,E2 -18462.698} C_VEL
LIN {X 0,Y 257.166,Z 305.58,A -85,B 0,C 180,E1 -18465.048,E2 -18465.048} C_VEL
LIN {X 0,Y 258.874,Z 298.638,A -85,B 0,C 180,E1 -18467.375,E2 -18467.375} C_VEL
LIN {X 0,Y 260.884,Z 289.949,A -85,B 0,C 180,E1 -18469.677,E2 -18469.677} C_VEL
LIN {X 0,Y 262.94,Z 281.053,A -85,B 0,C 180,E1 -18471.562,E2 -18471.562} C_VEL
LIN {X 0,Y 265.154,Z 271.292,A -85,B 0,C 180,E1 -18473.22,E2 -18473.22} C_VEL
LIN {X 0,Y 265.544,Z 267.522,A -85,B 0,C 180,E1 -18473.804,E2 -18473.804} C_VEL
LIN {X 0,Y 265.028,Z 257.27,A -85,B 0,C 180,E1 -18475.336,E2 -18475.336} C_VEL
LIN {X 0,Y 263.711,Z 245.926,A -85,B 0,C 180,E1 -18476.802,E2 -18476.802} C_VEL
LIN {X 0,Y 261.309,Z 233.604,A -85,B 0,C 180,E1 -18478.183,E2 -18478.183} C_VEL
LIN {X 0,Y 258.04,Z 221.459,A -85,B 0,C 180,E1 -18479.36,E2 -18479.36} C_VEL
LIN {X 0,Y 256.679,Z 216.267,A -85,B 0,C 180,E1 -18479.831,E2 -18479.831} C_VEL
LIN {X 0,Y 257.602,Z 211.513,A -85,B 0,C 180,E1 -18484.005,E2 -18484.005} C_VEL
LIN {X 0,Y 257.889,Z 208.443,A -85,B 0,C 180,E1 -18486.836,E2 -18486.836} C_VEL
LIN {X 0,Y 257.862,Z 206.407,A -85,B 0,C 180,E1 -18488.817,E2 -18488.817} C_VEL
LIN {X 0,Y 257.388,Z 202.817,A -85,B 0,C 180,E1 -18492.504,E2 -18492.504} C_VEL
LIN {X 0,Y 256.662,Z 198.946,A -85,B 0,C 180,E1 -18496.799,E2 -18496.799} C_VEL
LIN {X 0,Y 256.085,Z 195.588,A -85,B 0,C 180,E1 -18500.86,E2 -18500.86} C_VEL
LIN {X 0,Y 256.072,Z 195.591,A -85,B 0,C 180,E1 -18504.806,E2 -18504.806} C_VEL
LIN {X 0,Y 256.072,Z 195.591,A -85,B 0,C 180,E1 -18508.57,E2 -18508.57} C_VEL
LIN {X 0,Y 256.116,Z 195.582,A -85,B 0,C 180,E1 -18512.193,E2 -18512.193} C_VEL
LIN {X 0,Y 256.162,Z 195.576,A -85,B 0,C 180,E1 -18515.699,E2 -18515.699} C_VEL
LIN {X 0,Y 256.226,Z 195.569,A -85,B 0,C 180,E1 -18519.11,E2 -18519.11} C_VEL
LIN {X 0,Y 256.28,Z 195.561,A -85,B 0,C 180,E1 -18524.084,E2 -18524.084} C_VEL
LIN {X 0,Y 256.283,Z 195.562,A -85,B 0,C 180,E1 -18528.933,E2 -18528.933} C_VEL
LIN {X 0,Y 256.502,Z 195.535,A -85,B 0,C 180,E1 -18532.126,E2 -18532.126} C_VEL
LIN {X 0,Y 256.481,Z 195.536,A -85,B 0,C 180,E1 -18536.859,E2 -18536.859} C_VEL
LIN {X 0,Y 256.727,Z 195.507,A -85,B 0,C 180,E1 -18540,E2 -18540} C_VEL
LIN {X 0,Y 256.516,Z 195.53,A -85,B 0,C 180,E1 -18543.142,E2 -18543.142} C_VEL
LIN {X 0,Y 256.498,Z 195.536,A -85,B 0,C 180,E1 -18547.875,E2 -18547.875} C_VEL
LIN {X 0,Y 256.248,Z 195.564,A -85,B 0,C 180,E1 -18552.675,E2 -18552.675} C_VEL
LIN {X 0,Y 256.248,Z 195.565,A -85,B 0,C 180,E1 -18556.285,E2 -18556.285} C_VEL
LIN {X 0,Y 256.155,Z 195.576,A -85,B 0,C 180,E1 -18560.897,E2 -18560.897} C_VEL
LIN {X 0,Y 256.177,Z 195.575,A -85,B 0,C 180,E1 -18565.139,E2 -18565.139} C_VEL
LIN {X 0,Y 256.094,Z 195.585,A -85,B 0,C 180,E1 -18569.603,E2 -18569.603} C_VEL
LIN {X 0,Y 256.06,Z 195.59,A -85,B 0,C 180,E1 -18573.295,E2 -18573.295} C_VEL
LIN {X 0,Y 256.106,Z 195.582,A -85,B 0,C 180,E1 -18577.272,E2 -18577.272} C_VEL
LIN {X 0,Y 256.048,Z 195.59,A -85,B 0,C 180,E1 -18581.205,E2 -18581.205} C_VEL
LIN {X 0,Y 256.021,Z 195.596,A -85,B 0,C 180,E1 -18585.539,E2 -18585.539} C_VEL
LIN {X 0,Y 256.048,Z 195.795,A -85,B 0,C 180,E1 -18586.673,E2 -18586.673} C_VEL
LIN {X 0,Y 256.39,Z 198.29,A -85,B 0,C 180,E1 -18590.132,E2 -18590.132} C_VEL
LIN {X 0,Y 256.392,Z 200.455,A -85,B 0,C 180,E1 -18592.913,E2 -18592.913} C_VEL
LIN {X 0,Y 255.988,Z 203.548,A -85,B 0,C 180,E1 -18596.697,E2 -18596.697} C_VEL
LIN {X 0,Y 255.871,Z 204.769,A -85,B 0,C 180,E1 -18598.157,E2 -18598.157} C_VEL
LIN {X 0,Y 256.883,Z 207.962,A -85,B 0,C 180,E1 -18598.476,E2 -18598.476} C_VEL
LIN {X 0,Y 260.977,Z 219.393,A -85,B 0,C 180,E1 -18599.711,E2 -18599.711} C_VEL
LIN {X 0,Y 264.175,Z 231.172,A -85,B 0,C 180,E1 -18601.119,E2 -18601.119} C_VEL
LIN {X 0,Y 266.276,Z 242.027,A -85,B 0,C 180,E1 -18602.582,E2 -18602.582} C_VEL
LIN {X 0,Y 267.42,Z 251.443,A -85,B 0,C 180,E1 -18604.018,E2 -18604.018} C_VEL
LIN {X 0,Y 265.395,Z 261.732,A -85,B 0,C 180,E1 -18605.559,E2 -18605.559} C_VEL
LIN {X 0,Y 263.379,Z 270.754,A -85,B 0,C 180,E1 -18607.238,E2 -18607.238} C_VEL
LIN {X 0,Y 261.398,Z 279.018,A -85,B 0,C 180,E1 -18609.131,E2 -18609.131} C_VEL
LIN {X 0,Y 259.63,Z 285.87,A -85,B 0,C 180,E1 -18611.045,E2 -18611.045} C_VEL
LIN {X 0,Y 258.075,Z 292.58,A -85,B 0,C 180,E1 -18613.385,E2 -18613.385} C_VEL
LIN {X 0,Y 256.588,Z 297.935,A -85,B 0,C 180,E1 -18615.729,E2 -18615.729} C_VEL
LIN {X 0,Y 255.536,Z 302.11,A -85,B 0,C 180,E1 -18618.096,E2 -18618.096} C_VEL
LIN {X 0,Y 254.815,Z 305.226,A -85,B 0,C 180,E1 -18620.474,E2 -18620.474} C_VEL
LIN {X 0,Y 254.45,Z 306.775,A -85,B 0,C 180,E1 -18622.061,E2 -18622.061} C_VEL
LIN {X 0,Y 254.204,Z 308.293,A -85,B 0,C 180,E1 -18624.447,E2 -18624.447} C_VEL
LIN {X 0,Y 254.081,Z 308.919,A -85,B 0,C 180,E1 -18626.828,E2 -18626.828} C_VEL
LIN {X 0,Y 254.074,Z 308.862,A -85,B 0,C 180,E1 -18628.414,E2 -18628.414} C_VEL
LIN {X 0,Y 254.064,Z 308.411,A -85,B 0,C 180,E1 -18629.999,E2 -18629.999} C_VEL
LIN {X 0,Y 254.374,Z 306.271,A -85,B 0,C 180,E1 -18633.166,E2 -18633.166} C_VEL
LIN {X 0,Y 254.846,Z 303.597,A -85,B 0,C 180,E1 -18635.537,E2 -18635.537} C_VEL
LIN {X 0,Y 255.439,Z 299.923,A -85,B 0,C 180,E1 -18637.905,E2 -18637.905} C_VEL
LIN {X 0,Y 256.36,Z 295.139,A -85,B 0,C 180,E1 -18640.263,E2 -18640.263} C_VEL
LIN {X 0,Y 257.586,Z 289.103,A -85,B 0,C 180,E1 -18642.606,E2 -18642.606} C_VEL
LIN {X 0,Y 259.323,Z 281.591,A -85,B 0,C 180,E1 -18644.917,E2 -18644.917} C_VEL
LIN {X 0,Y 260.905,Z 273.914,A -85,B 0,C 180,E1 -18646.83,E2 -18646.83} C_VEL
LIN {X 0,Y 262.881,Z 263.482,A -85,B 0,C 180,E1 -18648.912,E2 -18648.912} C_VEL
LIN {X 0,Y 264.662,Z 253.419,A -85,B 0,C 180,E1 -18650.509,E2 -18650.509} C_VEL
LIN {X 0,Y 265.482,Z 247.568,A -85,B 0,C 180,E1 -18651.302,E2 -18651.302} C_VEL
LIN {X 0,Y 263.999,Z 236.741,A -85,B 0,C 180,E1 -18652.795,E2 -18652.795} C_VEL
LIN {X 0,Y 261.486,Z 224.435,A -85,B 0,C 180,E1 -18654.238,E2 -18654.238} C_VEL
LIN {X 0,Y 258.05,Z 212.47,A -85,B 0,C 180,E1 -18655.456,E2 -18655.456} C_VEL
LIN {X 0,Y 255.512,Z 204.635,A -85,B 0,C 180,E1 -18656.161,E2 -18656.161} C_VEL
LIN {X 0,Y 255.873,Z 201.631,A -85,B 0,C 180,E1 -18659.627,E2 -18659.627} C_VEL
LIN {X 0,Y 256.128,Z 198.558,A -85,B 0,C 180,E1 -18663.28,E2 -18663.28} C_VEL
LIN {X 0,Y 256.163,Z 197.038,A -85,B 0,C 180,E1 -18665.176,E2 -18665.176} C_VEL
LIN {X 0,Y 256.054,Z 195.595,A -85,B 0,C 180,E1 -18667.252,E2 -18667.252} C_VEL
LIN {X 0,Y 256.049,Z 195.591,A -85,B 0,C 180,E1 -18671.199,E2 -18671.199} C_VEL
LIN {X 0,Y 256.065,Z 195.588,A -85,B 0,C 180,E1 -18675.523,E2 -18675.523} C_VEL
LIN {X 0,Y 256.118,Z 195.583,A -85,B 0,C 180,E1 -18678.808,E2 -18678.808} C_VEL
LIN {X 0,Y 256.135,Z 195.58,A -85,B 0,C 180,E1 -18682.868,E2 -18682.868} C_VEL
LIN {X 0,Y 256.052,Z 195.592,A -85,B 0,C 180,E1 -18686.704,E2 -18686.704} C_VEL
LIN {X 0,Y 256.086,Z 195.586,A -85,B 0,C 180,E1 -18690.396,E2 -18690.396} C_VEL
LIN {X 0,Y 256.172,Z 195.571,A -85,B 0,C 180,E1 -18694.858,E2 -18694.858} C_VEL
LIN {X 0,Y 256.218,Z 195.539,A -85,B 0,C 180,E1 -18699.109,E2 -18699.109} C_VEL
LIN {X 0,Y 256.272,Z 195.56,A -85,B 0,C 180,E1 -18704.083,E2 -18704.083} C_VEL
LIN {X 0,Y 256.344,Z 195.544,A -85,B 0,C 180,E1 -18708.935,E2 -18708.935} C_VEL
LIN {X 0,Y 256.526,Z 195.533,A -85,B 0,C 180,E1 -18712.126,E2 -18712.126} C_VEL
LIN {X 0,Y 256.688,Z 195.509,A -85,B 0,C 180,E1 -18718.431,E2 -18718.431} C_VEL
LIN {X 0,Y 256.696,Z 195.51,A -85,B 0,C 180,E1 -18721.569,E2 -18721.569} C_VEL
LIN {X 0,Y 256.515,Z 195.533,A -85,B 0,C 180,E1 -18727.873,E2 -18727.873} C_VEL
LIN {X 0,Y 256.286,Z 195.562,A -85,B 0,C 180,E1 -18731.067,E2 -18731.067} C_VEL
LIN {X 0,Y 256.241,Z 195.566,A -85,B 0,C 180,E1 -18735.918,E2 -18735.918} C_VEL
LIN {X 0,Y 256.217,Z 195.572,A -85,B 0,C 180,E1 -18740.891,E2 -18740.891} C_VEL
LIN {X 0,Y 256.171,Z 195.577,A -85,B 0,C 180,E1 -18745.141,E2 -18745.141} C_VEL
LIN {X 0,Y 256.095,Z 195.577,A -85,B 0,C 180,E1 -18749.602,E2 -18749.602} C_VEL
LIN {X 0,Y 256.069,Z 195.58,A -85,B 0,C 180,E1 -18751.345,E2 -18751.345} C_VEL
LIN {X 0,Y 255.455,Z 195.664,A -85,B 0,C 180,E1 -18752.658,E2 -18752.658} C_VEL
LIN {X 0,Y 252.616,Z 196.02,A -85,B 0,C 180,E1 -18754.798,E2 -18754.798} C_VEL
LIN {X 0,Y 250.171,Z 196.324,A -85,B 0,C 180,E1 -18756.54,E2 -18756.54} C_VEL
LIN {X 0,Y 249.121,Z 196.454,A -85,B 0,C 180,E1 -18757.892,E2 -18757.892} C_VEL
LIN {X 0,Y 249.037,Z 196.465,A -85,B 0,C 180,E1 -18758.35,E2 -18758.35} C_VEL
LIN {X 0,Y 249.137,Z 196.579,A -85,B 0,C 180,E1 -18761.523,E2 -18761.523} C_VEL
LIN {X 0,Y 249.702,Z 199.874,A -85,B 0,C 180,E1 -18765.286,E2 -18765.286} C_VEL
LIN {X 0,Y 250.369,Z 204.116,A -85,B 0,C 180,E1 -18769.793,E2 -18769.793} C_VEL
LIN {X 0,Y 250.643,Z 207.281,A -85,B 0,C 180,E1 -18772.93,E2 -18772.93} C_VEL
LIN {X 0,Y 250.339,Z 210.401,A -85,B 0,C 180,E1 -18775.846,E2 -18775.846} C_VEL
LIN {X 0,Y 249.507,Z 214.521,A -85,B 0,C 180,E1 -18779.538,E2 -18779.538} C_VEL
LIN {X 0,Y 249.178,Z 216.306,A -85,B 0,C 180,E1 -18781.114,E2 -18781.114} C_VEL
LIN {X 0,Y 252.65,Z 230.004,A -85,B 0,C 180,E1 -18782.283,E2 -18782.283} C_VEL
LIN {X 0,Y 255.101,Z 242.959,A -85,B 0,C 180,E1 -18783.631,E2 -18783.631} C_VEL
LIN {X 0,Y 256.378,Z 254.299,A -85,B 0,C 180,E1 -18785.014,E2 -18785.014} C_VEL
LIN {X 0,Y 256.935,Z 265.557,A -85,B 0,C 180,E1 -18786.636,E2 -18786.636} C_VEL
LIN {X 0,Y 256.649,Z 269.476,A -85,B 0,C 180,E1 -18787.248,E2 -18787.248} C_VEL
LIN {X 0,Y 254.615,Z 279.6,A -85,B 0,C 180,E1 -18788.974,E2 -18788.974} C_VEL
LIN {X 0,Y 252.667,Z 289.168,A -85,B 0,C 180,E1 -18791.036,E2 -18791.036} C_VEL
LIN {X 0,Y 251.194,Z 296.297,A -85,B 0,C 180,E1 -18792.918,E2 -18792.918} C_VEL
LIN {X 0,Y 249.595,Z 303.709,A -85,B 0,C 180,E1 -18795.322,E2 -18795.322} C_VEL
LIN {X 0,Y 248.383,Z 309.659,A -85,B 0,C 180,E1 -18797.75,E2 -18797.75} C_VEL
LIN {X 0,Y 247.602,Z 314.357,A -85,B 0,C 180,E1 -18800.196,E2 -18800.196} C_VEL
LIN {X 0,Y 247.118,Z 317.94,A -85,B 0,C 180,E1 -18802.649,E2 -18802.649} C_VEL
LIN {X 0,Y 246.881,Z 320.511,A -85,B 0,C 180,E1 -18805.102,E2 -18805.102} C_VEL
LIN {X 0,Y 246.864,Z 321.72,A -85,B 0,C 180,E1 -18806.737,E2 -18806.737} C_VEL
LIN {X 0,Y 246.928,Z 322.488,A -85,B 0,C 180,E1 -18808.37,E2 -18808.37} C_VEL
LIN {X 0,Y 246.982,Z 322.855,A -85,B 0,C 180,E1 -18810.001,E2 -18810.001} C_VEL
LIN {X 0,Y 246.921,Z 322.831,A -85,B 0,C 180,E1 -18811.632,E2 -18811.632} C_VEL
LIN {X 0,Y 246.853,Z 322.421,A -85,B 0,C 180,E1 -18813.265,E2 -18813.265} C_VEL
LIN {X 0,Y 246.882,Z 321.584,A -85,B 0,C 180,E1 -18814.9,E2 -18814.9} C_VEL
LIN {X 0,Y 247.268,Z 318.685,A -85,B 0,C 180,E1 -18818.171,E2 -18818.171} C_VEL
LIN {X 0,Y 247.892,Z 315.375,A -85,B 0,C 180,E1 -18820.62,E2 -18820.62} C_VEL
LIN {X 0,Y 248.83,Z 311.001,A -85,B 0,C 180,E1 -18823.059,E2 -18823.059} C_VEL
LIN {X 0,Y 250.291,Z 305.445,A -85,B 0,C 180,E1 -18825.471,E2 -18825.471} C_VEL
LIN {X 0,Y 252.092,Z 298.519,A -85,B 0,C 180,E1 -18827.858,E2 -18827.858} C_VEL
LIN {X 0,Y 254.183,Z 289.853,A -85,B 0,C 180,E1 -18830.218,E2 -18830.218} C_VEL
LIN {X 0,Y 256.34,Z 280.978,A -85,B 0,C 180,E1 -18832.146,E2 -18832.146} C_VEL
LIN {X 0,Y 258.834,Z 270.059,A -85,B 0,C 180,E1 -18834.034,E2 -18834.034} C_VEL
LIN {X 0,Y 258.58,Z 260.613,A -85,B 0,C 180,E1 -18835.555,E2 -18835.555} C_VEL
LIN {X 0,Y 257.424,Z 248.779,A -85,B 0,C 180,E1 -18837.201,E2 -18837.201} C_VEL
LIN {X 0,Y 255.477,Z 237.563,A -85,B 0,C 180,E1 -18838.563,E2 -18838.563} C_VEL
LIN {X 0,Y 252.4,Z 225.097,A -85,B 0,C 180,E1 -18839.891,E2 -18839.891} C_VEL
LIN {X 0,Y 249.822,Z 216.062,A -85,B 0,C 180,E1 -18840.772,E2 -18840.772} C_VEL
LIN {X 0,Y 250.595,Z 212.352,A -85,B 0,C 180,E1 -18844.117,E2 -18844.117} C_VEL
LIN {X 0,Y 250.88,Z 209.315,A -85,B 0,C 180,E1 -18847.032,E2 -18847.032} C_VEL
LIN {X 0,Y 250.709,Z 206.241,A -85,B 0,C 180,E1 -18850.145,E2 -18850.145} C_VEL
LIN {X 0,Y 250.302,Z 203.481,A -85,B 0,C 180,E1 -18853.111,E2 -18853.111} C_VEL
LIN {X 0,Y 249.61,Z 199.687,A -85,B 0,C 180,E1 -18857.488,E2 -18857.488} C_VEL
LIN {X 0,Y 249.028,Z 196.467,A -85,B 0,C 180,E1 -18861.62,E2 -18861.62} C_VEL
LIN {X 0,Y 249.034,Z 196.469,A -85,B 0,C 180,E1 -18865.638,E2 -18865.638} C_VEL
LIN {X 0,Y 248.996,Z 196.473,A -85,B 0,C 180,E1 -18869.466,E2 -18869.466} C_VEL
LIN {X 0,Y 249.057,Z 196.464,A -85,B 0,C 180,E1 -18873.161,E2 -18873.161} C_VEL
LIN {X 0,Y 249.091,Z 196.459,A -85,B 0,C 180,E1 -18876.734,E2 -18876.734} C_VEL
LIN {X 0,Y 249.135,Z 196.452,A -85,B 0,C 180,E1 -18880.214,E2 -18880.214} C_VEL
LIN {X 0,Y 249.231,Z 196.439,A -85,B 0,C 180,E1 -18883.621,E2 -18883.621} C_VEL
LIN {X 0,Y 249.23,Z 196.441,A -85,B 0,C 180,E1 -18888.616,E2 -18888.616} C_VEL
LIN {X 0,Y 249.441,Z 196.413,A -85,B 0,C 180,E1 -18891.902,E2 -18891.902} C_VEL
LIN {X 0,Y 249.28,Z 196.431,A -85,B 0,C 180,E1 -18895.148,E2 -18895.148} C_VEL
LIN {X 0,Y 249.658,Z 196.387,A -85,B 0,C 180,E1 -18898.387,E2 -18898.387} C_VEL
LIN {X 0,Y 249.669,Z 196.384,A -85,B 0,C 180,E1 -18901.613,E2 -18901.613} C_VEL
LIN {X 0,Y 249.426,Z 196.413,A -85,B 0,C 180,E1 -18906.696,E2 -18906.696} C_VEL
LIN {X 0,Y 249.321,Z 196.428,A -85,B 0,C 180,E1 -18909.738,E2 -18909.738} C_VEL
LIN {X 0,Y 249.183,Z 196.443,A -85,B 0,C 180,E1 -18914.705,E2 -18914.705} C_VEL
LIN {X 0,Y 249.123,Z 196.453,A -85,B 0,C 180,E1 -18918.079,E2 -18918.079} C_VEL
LIN {X 0,Y 249.077,Z 196.46,A -85,B 0,C 180,E1 -18921.52,E2 -18921.52} C_VEL
LIN {X 0,Y 249.12,Z 196.455,A -85,B 0,C 180,E1 -18925.483,E2 -18925.483} C_VEL
LIN {X 0,Y 249.064,Z 196.461,A -85,B 0,C 180,E1 -18928.99,E2 -18928.99} C_VEL
LIN {X 0,Y 249.023,Z 196.465,A -85,B 0,C 180,E1 -18932.428,E2 -18932.428} C_VEL
LIN {X 0,Y 249.04,Z 196.464,A -85,B 0,C 180,E1 -18936.344,E2 -18936.344} C_VEL
LIN {X 0,Y 249,Z 196.468,A -85,B 0,C 180,E1 -18940.48,E2 -18940.48} C_VEL
LIN {X 0,Y 248.996,Z 196.471,A -85,B 0,C 180,E1 -18942.792,E2 -18942.792} C_VEL
LIN {X 0,Y 248.97,Z 196.473,A -85,B 0,C 180,E1 -18945.116,E2 -18945.116} C_VEL
LIN {X 0,Y 249.113,Z 197.52,A -85,B 0,C 180,E1 -18947.386,E2 -18947.386} C_VEL
LIN {X 0,Y 249.336,Z 199.045,A -85,B 0,C 180,E1 -18949.589,E2 -18949.589} C_VEL
LIN {X 0,Y 249.385,Z 200.917,A -85,B 0,C 180,E1 -18952.1,E2 -18952.1} C_VEL
LIN {X 0,Y 249.093,Z 203.744,A -85,B 0,C 180,E1 -18955.649,E2 -18955.649} C_VEL
LIN {X 0,Y 248.938,Z 205.003,A -85,B 0,C 180,E1 -18957.21,E2 -18957.21} C_VEL
LIN {X 0,Y 250.01,Z 208.255,A -85,B 0,C 180,E1 -18957.548,E2 -18957.548} C_VEL
LIN {X 0,Y 254.367,Z 220.322,A -85,B 0,C 180,E1 -18958.928,E2 -18958.928} C_VEL
LIN {X 0,Y 257.304,Z 231.023,A -85,B 0,C 180,E1 -18960.272,E2 -18960.272} C_VEL
LIN {X 0,Y 259.43,Z 241.592,A -85,B 0,C 180,E1 -18961.749,E2 -18961.749} C_VEL
LIN {X 0,Y 260.82,Z 252.554,A -85,B 0,C 180,E1 -18963.485,E2 -18963.485} C_VEL
LIN {X 0,Y 258.434,Z 263.908,A -85,B 0,C 180,E1 -18965.285,E2 -18965.285} C_VEL
LIN {X 0,Y 256.386,Z 272.599,A -85,B 0,C 180,E1 -18967.008,E2 -18967.008} C_VEL
LIN {X 0,Y 254.354,Z 280.588,A -85,B 0,C 180,E1 -18968.949,E2 -18968.949} C_VEL
LIN {X 0,Y 252.243,Z 288.432,A -85,B 0,C 180,E1 -18971.32,E2 -18971.32} C_VEL
LIN {X 0,Y 250.741,Z 294.643,A -85,B 0,C 180,E1 -18973.723,E2 -18973.723} C_VEL
LIN {X 0,Y 249.248,Z 299.598,A -85,B 0,C 180,E1 -18976.133,E2 -18976.133} C_VEL
LIN {X 0,Y 248.299,Z 303.424,A -85,B 0,C 180,E1 -18978.572,E2 -18978.572} C_VEL
LIN {X 0,Y 247.8,Z 305.391,A -85,B 0,C 180,E1 -18980.202,E2 -18980.202} C_VEL
LIN {X 0,Y 247.399,Z 306.946,A -85,B 0,C 180,E1 -18981.834,E2 -18981.834} C_VEL
LIN {X 0,Y 247.091,Z 308.614,A -85,B 0,C 180,E1 -18984.572,E2 -18984.572} C_VEL
LIN {X 0,Y 246.98,Z 309.114,A -85,B 0,C 180,E1 -18986.737,E2 -18986.737} C_VEL
LIN {X 0,Y 246.983,Z 309.062,A -85,B 0,C 180,E1 -18988.368,E2 -18988.368} C_VEL
LIN {X 0,Y 246.993,Z 308.622,A -85,B 0,C 180,E1 -18989.999,E2 -18989.999} C_VEL
LIN {X 0,Y 247.316,Z 306.495,A -85,B 0,C 180,E1 -18993.257,E2 -18993.257} C_VEL
LIN {X 0,Y 247.795,Z 303.834,A -85,B 0,C 180,E1 -18995.695,E2 -18995.695} C_VEL
LIN {X 0,Y 248.42,Z 300.174,A -85,B 0,C 180,E1 -18998.13,E2 -18998.13} C_VEL
LIN {X 0,Y 249.398,Z 295.404,A -85,B 0,C 180,E1 -19000.553,E2 -19000.553} C_VEL
LIN {X 0,Y 250.681,Z 289.384,A -85,B 0,C 180,E1 -19002.959,E2 -19002.959} C_VEL
LIN {X 0,Y 252.464,Z 281.89,A -85,B 0,C 180,E1 -19005.332,E2 -19005.332} C_VEL
LIN {X 0,Y 254.135,Z 274.235,A -85,B 0,C 180,E1 -19007.292,E2 -19007.292} C_VEL
LIN {X 0,Y 256.204,Z 263.838,A -85,B 0,C 180,E1 -19009.424,E2 -19009.424} C_VEL
LIN {X 0,Y 258.021,Z 253.952,A -85,B 0,C 180,E1 -19011.038,E2 -19011.038} C_VEL
LIN {X 0,Y 258.763,Z 248.594,A -85,B 0,C 180,E1 -19011.793,E2 -19011.793} C_VEL
LIN {X 0,Y 257.487,Z 238.845,A -85,B 0,C 180,E1 -19013.21,E2 -19013.21} C_VEL
LIN {X 0,Y 255.25,Z 227.169,A -85,B 0,C 180,E1 -19014.684,E2 -19014.684} C_VEL
LIN {X 0,Y 251.919,Z 215.093,A -85,B 0,C 180,E1 -19016.004,E2 -19016.004} C_VEL
LIN {X 0,Y 248.651,Z 205.319,A -85,B 0,C 180,E1 -19016.937,E2 -19016.937} C_VEL
LIN {X 0,Y 248.61,Z 204.832,A -85,B 0,C 180,E1 -19017.002,E2 -19017.002} C_VEL
LIN {X 0,Y 248.908,Z 201.833,A -85,B 0,C 180,E1 -19020.543,E2 -19020.543} C_VEL
LIN {X 0,Y 249.138,Z 198.771,A -85,B 0,C 180,E1 -19024.342,E2 -19024.342} C_VEL
LIN {X 0,Y 249.053,Z 197.266,A -85,B 0,C 180,E1 -19026.337,E2 -19026.337} C_VEL
LIN {X 0,Y 249.003,Z 196.473,A -85,B 0,C 180,E1 -19027.787,E2 -19027.787} C_VEL
LIN {X 0,Y 248.999,Z 196.469,A -85,B 0,C 180,E1 -19030.475,E2 -19030.475} C_VEL
LIN {X 0,Y 249.008,Z 196.47,A -85,B 0,C 180,E1 -19034.872,E2 -19034.872} C_VEL
LIN {X 0,Y 249.069,Z 196.462,A -85,B 0,C 180,E1 -19037.373,E2 -19037.373} C_VEL
LIN {X 0,Y 249.038,Z 196.463,A -85,B 0,C 180,E1 -19041.621,E2 -19041.621} C_VEL
LIN {X 0,Y 249.03,Z 196.464,A -85,B 0,C 180,E1 -19045.637,E2 -19045.637} C_VEL
LIN {X 0,Y 249.031,Z 196.464,A -85,B 0,C 180,E1 -19049.47,E2 -19049.47} C_VEL
LIN {X 0,Y 249.055,Z 196.461,A -85,B 0,C 180,E1 -19053.16,E2 -19053.16} C_VEL
LIN {X 0,Y 249.083,Z 196.442,A -85,B 0,C 180,E1 -19056.732,E2 -19056.732} C_VEL
LIN {X 0,Y 249.126,Z 196.424,A -85,B 0,C 180,E1 -19060.212,E2 -19060.212} C_VEL
LIN {X 0,Y 249.222,Z 196.435,A -85,B 0,C 180,E1 -19063.62,E2 -19063.62} C_VEL
LIN {X 0,Y 249.27,Z 196.426,A -85,B 0,C 180,E1 -19068.617,E2 -19068.617} C_VEL
LIN {X 0,Y 249.472,Z 196.409,A -85,B 0,C 180,E1 -19071.902,E2 -19071.902} C_VEL
LIN {X 0,Y 249.411,Z 196.409,A -85,B 0,C 180,E1 -19076.769,E2 -19076.769} C_VEL
LIN {X 0,Y 249.689,Z 196.383,A -85,B 0,C 180,E1 -19080,E2 -19080} C_VEL
LIN {X 0,Y 249.443,Z 196.413,A -85,B 0,C 180,E1 -19083.23,E2 -19083.23} C_VEL
LIN {X 0,Y 249.457,Z 196.411,A -85,B 0,C 180,E1 -19088.098,E2 -19088.098} C_VEL
LIN {X 0,Y 249.229,Z 196.442,A -85,B 0,C 180,E1 -19091.384,E2 -19091.384} C_VEL
LIN {X 0,Y 249.175,Z 196.446,A -85,B 0,C 180,E1 -19096.487,E2 -19096.487} C_VEL
LIN {X 0,Y 249.139,Z 196.452,A -85,B 0,C 180,E1 -19101.438,E2 -19101.438} C_VEL
LIN {X 0,Y 249.113,Z 196.454,A -85,B 0,C 180,E1 -19105.485,E2 -19105.485} C_VEL
LIN {X 0,Y 249.064,Z 196.455,A -85,B 0,C 180,E1 -19108.995,E2 -19108.995} C_VEL
LIN {X 0,Y 249.018,Z 196.463,A -85,B 0,C 180,E1 -19112.427,E2 -19112.427} C_VEL
LIN {X 0,Y 249.057,Z 196.463,A -85,B 0,C 180,E1 -19116.341,E2 -19116.341} C_VEL
LIN {X 0,Y 249.037,Z 196.465,A -85,B 0,C 180,E1 -19118.35,E2 -19118.35} C_VEL
LIN {X 0,Y 248.398,Z 196.74,A -85,B 0,C 180,E1 -19119.698,E2 -19119.698} C_VEL
LIN {X 0,Y 245.705,Z 198.081,A -85,B 0,C 180,E1 -19121.888,E2 -19121.888} C_VEL
LIN {X 0,Y 243.509,Z 199.627,A -85,B 0,C 180,E1 -19123.658,E2 -19123.658} C_VEL
LIN {X 0,Y 242.695,Z 200.876,A -85,B 0,C 180,E1 -19125.022,E2 -19125.022} C_VEL
LIN {X 0,Y 242.696,Z 201.284,A -85,B 0,C 180,E1 -19125.482,E2 -19125.482} C_VEL
LIN {X 0,Y 243.16,Z 204.217,A -85,B 0,C 180,E1 -19128.718,E2 -19128.718} C_VEL
LIN {X 0,Y 243.5,Z 206.57,A -85,B 0,C 180,E1 -19131.195,E2 -19131.195} C_VEL
LIN {X 0,Y 243.537,Z 209.29,A -85,B 0,C 180,E1 -19133.903,E2 -19133.903} C_VEL
LIN {X 0,Y 243.022,Z 212.558,A -85,B 0,C 180,E1 -19136.998,E2 -19136.998} C_VEL
LIN {X 0,Y 242.269,Z 216.076,A -85,B 0,C 180,E1 -19140.226,E2 -19140.226} C_VEL
LIN {X 0,Y 246.021,Z 230.577,A -85,B 0,C 180,E1 -19141.559,E2 -19141.559} C_VEL
LIN {X 0,Y 248.457,Z 243.534,A -85,B 0,C 180,E1 -19142.976,E2 -19142.976} C_VEL
LIN {X 0,Y 249.706,Z 254.846,A -85,B 0,C 180,E1 -19144.422,E2 -19144.422} C_VEL
LIN {X 0,Y 250.165,Z 266.496,A -85,B 0,C 180,E1 -19146.184,E2 -19146.184} C_VEL
LIN {X 0,Y 249.863,Z 270.364,A -85,B 0,C 180,E1 -19146.813,E2 -19146.813} C_VEL
LIN {X 0,Y 247.551,Z 281.237,A -85,B 0,C 180,E1 -19148.781,E2 -19148.781} C_VEL
LIN {X 0,Y 245.777,Z 289.575,A -85,B 0,C 180,E1 -19150.671,E2 -19150.671} C_VEL
LIN {X 0,Y 244.067,Z 297.374,A -85,B 0,C 180,E1 -19152.836,E2 -19152.836} C_VEL
LIN {X 0,Y 242.465,Z 304.554,A -85,B 0,C 180,E1 -19155.31,E2 -19155.31} C_VEL
LIN {X 0,Y 241.406,Z 309.402,A -85,B 0,C 180,E1 -19157.39,E2 -19157.39} C_VEL
LIN {X 0,Y 240.587,Z 314.114,A -85,B 0,C 180,E1 -19159.907,E2 -19159.907} C_VEL
LIN {X 0,Y 240.049,Z 317.708,A -85,B 0,C 180,E1 -19162.431,E2 -19162.431} C_VEL
LIN {X 0,Y 239.773,Z 320.551,A -85,B 0,C 180,E1 -19165.257,E2 -19165.257} C_VEL
LIN {X 0,Y 239.837,Z 322.283,A -85,B 0,C 180,E1 -19168.322,E2 -19168.322} C_VEL
LIN {X 0,Y 239.891,Z 322.654,A -85,B 0,C 180,E1 -19170.001,E2 -19170.001} C_VEL
LIN {X 0,Y 239.83,Z 322.636,A -85,B 0,C 180,E1 -19171.68,E2 -19171.68} C_VEL
LIN {X 0,Y 239.79,Z 321.561,A -85,B 0,C 180,E1 -19174.793,E2 -19174.793} C_VEL
LIN {X 0,Y 239.952,Z 320.16,A -85,B 0,C 180,E1 -19176.729,E2 -19176.729} C_VEL
LIN {X 0,Y 240.415,Z 317.53,A -85,B 0,C 180,E1 -19179.253,E2 -19179.253} C_VEL
LIN {X 0,Y 241.2,Z 313.891,A -85,B 0,C 180,E1 -19181.769,E2 -19181.769} C_VEL
LIN {X 0,Y 242.353,Z 309.148,A -85,B 0,C 180,E1 -19184.27,E2 -19184.27} C_VEL
LIN {X 0,Y 244.383,Z 302.042,A -85,B 0,C 180,E1 -19187.144,E2 -19187.144} C_VEL
LIN {X 0,Y 246.332,Z 294.579,A -85,B 0,C 180,E1 -19189.511,E2 -19189.511} C_VEL
LIN {X 0,Y 248.378,Z 286.439,A -85,B 0,C 180,E1 -19191.582,E2 -19191.582} C_VEL
LIN {X 0,Y 250.795,Z 276.826,A -85,B 0,C 180,E1 -19193.535,E2 -19193.535} C_VEL
LIN {X 0,Y 252.19,Z 270.014,A -85,B 0,C 180,E1 -19194.709,E2 -19194.709} C_VEL
LIN {X 0,Y 251.829,Z 259.022,A -85,B 0,C 180,E1 -19196.52,E2 -19196.52} C_VEL
LIN {X 0,Y 250.606,Z 247.479,A -85,B 0,C 180,E1 -19198.161,E2 -19198.161} C_VEL
LIN {X 0,Y 248.336,Z 235.263,A -85,B 0,C 180,E1 -19199.685,E2 -19199.685} C_VEL
LIN {X 0,Y 245.03,Z 222.693,A -85,B 0,C 180,E1 -19201.064,E2 -19201.064} C_VEL
LIN {X 0,Y 243.048,Z 216.535,A -85,B 0,C 180,E1 -19201.675,E2 -19201.675} C_VEL
LIN {X 0,Y 242.974,Z 215.873,A -85,B 0,C 180,E1 -19201.739,E2 -19201.739} C_VEL
LIN {X 0,Y 243.678,Z 212.213,A -85,B 0,C 180,E1 -19205.226,E2 -19205.226} C_VEL
LIN {X 0,Y 243.876,Z 210.174,A -85,B 0,C 180,E1 -19207.24,E2 -19207.24} C_VEL
LIN {X 0,Y 243.753,Z 208.103,A -85,B 0,C 180,E1 -19209.367,E2 -19209.367} C_VEL
LIN {X 0,Y 243.51,Z 206.061,A -85,B 0,C 180,E1 -19211.589,E2 -19211.589} C_VEL
LIN {X 0,Y 243.169,Z 204.015,A -85,B 0,C 180,E1 -19213.916,E2 -19213.916} C_VEL
LIN {X 0,Y 242.495,Z 200.469,A -85,B 0,C 180,E1 -19218.196,E2 -19218.196} C_VEL
LIN {X 0,Y 242.015,Z 197.341,A -85,B 0,C 180,E1 -19222.322,E2 -19222.322} C_VEL
LIN {X 0,Y 241.97,Z 197.347,A -85,B 0,C 180,E1 -19226.506,E2 -19226.506} C_VEL
LIN {X 0,Y 241.976,Z 197.346,A -85,B 0,C 180,E1 -19230.608,E2 -19230.608} C_VEL
LIN {X 0,Y 242.058,Z 197.333,A -85,B 0,C 180,E1 -19234.182,E2 -19234.182} C_VEL
LIN {X 0,Y 242.077,Z 197.331,A -85,B 0,C 180,E1 -19238.276,E2 -19238.276} C_VEL
LIN {X 0,Y 242.152,Z 197.321,A -85,B 0,C 180,E1 -19243.278,E2 -19243.278} C_VEL
LIN {X 0,Y 242.166,Z 197.319,A -85,B 0,C 180,E1 -19248.279,E2 -19248.279} C_VEL
LIN {X 0,Y 242.387,Z 197.291,A -85,B 0,C 180,E1 -19251.665,E2 -19251.665} C_VEL
LIN {X 0,Y 242.241,Z 197.308,A -85,B 0,C 180,E1 -19255.007,E2 -19255.007} C_VEL
LIN {X 0,Y 242.619,Z 197.264,A -85,B 0,C 180,E1 -19258.34,E2 -19258.34} C_VEL
LIN {X 0,Y 242.631,Z 197.261,A -85,B 0,C 180,E1 -19261.66,E2 -19261.66} C_VEL
LIN {X 0,Y 242.407,Z 197.288,A -85,B 0,C 180,E1 -19266.666,E2 -19266.666} C_VEL
LIN {X 0,Y 242.25,Z 197.31,A -85,B 0,C 180,E1 -19270.025,E2 -19270.025} C_VEL
LIN {X 0,Y 242.138,Z 197.321,A -85,B 0,C 180,E1 -19275.143,E2 -19275.143} C_VEL
LIN {X 0,Y 242.059,Z 197.332,A -85,B 0,C 180,E1 -19278.626,E2 -19278.626} C_VEL
LIN {X 0,Y 242.003,Z 197.339,A -85,B 0,C 180,E1 -19282.182,E2 -19282.182} C_VEL
LIN {X 0,Y 242.058,Z 197.332,A -85,B 0,C 180,E1 -19285.84,E2 -19285.84} C_VEL
LIN {X 0,Y 241.999,Z 197.341,A -85,B 0,C 180,E1 -19289.585,E2 -19289.585} C_VEL
LIN {X 0,Y 241.973,Z 197.344,A -85,B 0,C 180,E1 -19293.494,E2 -19293.494} C_VEL
LIN {X 0,Y 241.982,Z 197.341,A -85,B 0,C 180,E1 -19297.584,E2 -19297.584} C_VEL
LIN {X 0,Y 241.928,Z 197.348,A -85,B 0,C 180,E1 -19301.925,E2 -19301.925} C_VEL
LIN {X 0,Y 241.909,Z 197.353,A -85,B 0,C 180,E1 -19304.208,E2 -19304.208} C_VEL
LIN {X 0,Y 241.963,Z 197.69,A -85,B 0,C 180,E1 -19305.808,E2 -19305.808} C_VEL
LIN {X 0,Y 242.246,Z 199.818,A -85,B 0,C 180,E1 -19308.966,E2 -19308.966} C_VEL
LIN {X 0,Y 242.338,Z 202.32,A -85,B 0,C 180,E1 -19312.483,E2 -19312.483} C_VEL
LIN {X 0,Y 242.008,Z 205.203,A -85,B 0,C 180,E1 -19316.183,E2 -19316.183} C_VEL
LIN {X 0,Y 243.078,Z 208.478,A -85,B 0,C 180,E1 -19316.545,E2 -19316.545} C_VEL
LIN {X 0,Y 247.551,Z 220.541,A -85,B 0,C 180,E1 -19318.012,E2 -19318.012} C_VEL
LIN {X 0,Y 250.765,Z 231.925,A -85,B 0,C 180,E1 -19319.523,E2 -19319.523} C_VEL
LIN {X 0,Y 252.933,Z 243.053,A -85,B 0,C 180,E1 -19321.157,E2 -19321.157} C_VEL
LIN {X 0,Y 254.203,Z 253.617,A -85,B 0,C 180,E1 -19322.92,E2 -19322.92} C_VEL
LIN {X 0,Y 251.741,Z 265.016,A -85,B 0,C 180,E1 -19324.803,E2 -19324.803} C_VEL
LIN {X 0,Y 249.412,Z 274.423,A -85,B 0,C 180,E1 -19326.766,E2 -19326.766} C_VEL
LIN {X 0,Y 246.926,Z 283.471,A -85,B 0,C 180,E1 -19329.16,E2 -19329.16} C_VEL
LIN {X 0,Y 244.898,Z 290.753,A -85,B 0,C 180,E1 -19331.599,E2 -19331.599} C_VEL
LIN {X 0,Y 243.355,Z 296.576,A -85,B 0,C 180,E1 -19334.076,E2 -19334.076} C_VEL
LIN {X 0,Y 241.911,Z 301.16,A -85,B 0,C 180,E1 -19336.56,E2 -19336.56} C_VEL
LIN {X 0,Y 241.297,Z 303.583,A -85,B 0,C 180,E1 -19338.236,E2 -19338.236} C_VEL
LIN {X 0,Y 240.772,Z 305.556,A -85,B 0,C 180,E1 -19339.913,E2 -19339.913} C_VEL
LIN {X 0,Y 240.369,Z 307.117,A -85,B 0,C 180,E1 -19341.593,E2 -19341.593} C_VEL
LIN {X 0,Y 239.987,Z 308.9,A -85,B 0,C 180,E1 -19344.684,E2 -19344.684} C_VEL
LIN {X 0,Y 239.883,Z 309.309,A -85,B 0,C 180,E1 -19346.64,E2 -19346.64} C_VEL
LIN {X 0,Y 239.893,Z 309.263,A -85,B 0,C 180,E1 -19348.32,E2 -19348.32} C_VEL
LIN {X 0,Y 239.924,Z 308.831,A -85,B 0,C 180,E1 -19349.999,E2 -19349.999} C_VEL
LIN {X 0,Y 240.237,Z 306.719,A -85,B 0,C 180,E1 -19353.353,E2 -19353.353} C_VEL
LIN {X 0,Y 240.746,Z 304.071,A -85,B 0,C 180,E1 -19355.863,E2 -19355.863} C_VEL
LIN {X 0,Y 241.408,Z 300.424,A -85,B 0,C 180,E1 -19358.368,E2 -19358.368} C_VEL
LIN {X 0,Y 242.416,Z 295.669,A -85,B 0,C 180,E1 -19360.86,E2 -19360.86} C_VEL
LIN {X 0,Y 243.768,Z 289.664,A -85,B 0,C 180,E1 -19363.333,E2 -19363.333} C_VEL
LIN {X 0,Y 245.624,Z 282.189,A -85,B 0,C 180,E1 -19365.77,E2 -19365.77} C_VEL
LIN {X 0,Y 247.388,Z 274.553,A -85,B 0,C 180,E1 -19367.779,E2 -19367.779} C_VEL
LIN {X 0,Y 249.544,Z 264.193,A -85,B 0,C 180,E1 -19369.964,E2 -19369.964} C_VEL
LIN {X 0,Y 251.407,Z 254.479,A -85,B 0,C 180,E1 -19371.596,E2 -19371.596} C_VEL
LIN {X 0,Y 252.068,Z 251.228,A -85,B 0,C 180,E1 -19372.062,E2 -19372.062} C_VEL
LIN {X 0,Y 251.153,Z 241.95,A -85,B 0,C 180,E1 -19373.497,E2 -19373.497} C_VEL
LIN {X 0,Y 249.147,Z 230.691,A -85,B 0,C 180,E1 -19375.029,E2 -19375.029} C_VEL
LIN {X 0,Y 246.15,Z 218.876,A -85,B 0,C 180,E1 -19376.434,E2 -19376.434} C_VEL
LIN {X 0,Y 241.726,Z 205.503,A -85,B 0,C 180,E1 -19377.814,E2 -19377.814} C_VEL
LIN {X 0,Y 241.671,Z 205.029,A -85,B 0,C 180,E1 -19377.843,E2 -19377.843} C_VEL
LIN {X 0,Y 242.023,Z 201.18,A -85,B 0,C 180,E1 -19382.634,E2 -19382.634} C_VEL
LIN {X 0,Y 242.103,Z 198.914,A -85,B 0,C 180,E1 -19385.628,E2 -19385.628} C_VEL
LIN {X 0,Y 241.96,Z 197.505,A -85,B 0,C 180,E1 -19387.583,E2 -19387.583} C_VEL
LIN {X 0,Y 241.934,Z 197.349,A -85,B 0,C 180,E1 -19391.918,E2 -19391.918} C_VEL
LIN {X 0,Y 241.991,Z 197.342,A -85,B 0,C 180,E1 -19396.551,E2 -19396.551} C_VEL
LIN {X 0,Y 241.998,Z 197.34,A -85,B 0,C 180,E1 -19400.288,E2 -19400.288} C_VEL
LIN {X 0,Y 241.981,Z 197.343,A -85,B 0,C 180,E1 -19404.487,E2 -19404.487} C_VEL
LIN {X 0,Y 241.957,Z 197.344,A -85,B 0,C 180,E1 -19408.477,E2 -19408.477} C_VEL
LIN {X 0,Y 241.986,Z 197.341,A -85,B 0,C 180,E1 -19412.309,E2 -19412.309} C_VEL
LIN {X 0,Y 242.052,Z 197.324,A -85,B 0,C 180,E1 -19416.015,E2 -19416.015} C_VEL
LIN {X 0,Y 242.062,Z 197.299,A -85,B 0,C 180,E1 -19419.61,E2 -19419.61} C_VEL
LIN {X 0,Y 242.144,Z 197.316,A -85,B 0,C 180,E1 -19423.276,E2 -19423.276} C_VEL
LIN {X 0,Y 242.194,Z 197.309,A -85,B 0,C 180,E1 -19428.28,E2 -19428.28} C_VEL
LIN {X 0,Y 242.422,Z 197.286,A -85,B 0,C 180,E1 -19431.665,E2 -19431.665} C_VEL
LIN {X 0,Y 242.238,Z 197.305,A -85,B 0,C 180,E1 -19435.006,E2 -19435.006} C_VEL
LIN {X 0,Y 242.611,Z 197.263,A -85,B 0,C 180,E1 -19438.34,E2 -19438.34} C_VEL
LIN {X 0,Y 242.621,Z 197.264,A -85,B 0,C 180,E1 -19441.66,E2 -19441.66} C_VEL
LIN {X 0,Y 242.41,Z 197.287,A -85,B 0,C 180,E1 -19446.659,E2 -19446.659} C_VEL
LIN {X 0,Y 242.292,Z 197.304,A -85,B 0,C 180,E1 -19450.022,E2 -19450.022} C_VEL
LIN {X 0,Y 242.119,Z 197.328,A -85,B 0,C 180,E1 -19455.144,E2 -19455.144} C_VEL
LIN {X 0,Y 242.063,Z 197.333,A -85,B 0,C 180,E1 -19458.625,E2 -19458.625} C_VEL
LIN {X 0,Y 242.05,Z 197.334,A -85,B 0,C 180,E1 -19462.176,E2 -19462.176} C_VEL
LIN {X 0,Y 242.048,Z 197.333,A -85,B 0,C 180,E1 -19465.84,E2 -19465.84} C_VEL
LIN {X 0,Y 242.012,Z 197.33,A -85,B 0,C 180,E1 -19469.582,E2 -19469.582} C_VEL
LIN {X 0,Y 241.974,Z 197.342,A -85,B 0,C 180,E1 -19473.493,E2 -19473.493} C_VEL
LIN {X 0,Y 241.996,Z 197.341,A -85,B 0,C 180,E1 -19477.58,E2 -19477.58} C_VEL
LIN {X 0,Y 242.083,Z 197.481,A -85,B 0,C 180,E1 -19480.997,E2 -19480.997} C_VEL
LIN {X 0,Y 242.696,Z 201.284,A -85,B 0,C 180,E1 -19485.482,E2 -19485.482} C_VEL
LIN {X 0,Y 242.268,Z 202.6,A -85,B 0,C 180,E1 -19486.836,E2 -19486.836} C_VEL
LIN {X 0,Y 239.731,Z 205.076,A -85,B 0,C 180,E1 -19489.036,E2 -19489.036} C_VEL
LIN {X 0,Y 237.487,Z 207.128,A -85,B 0,C 180,E1 -19490.824,E2 -19490.824} C_VEL
LIN {X 0,Y 236.547,Z 208.605,A -85,B 0,C 180,E1 -19492.21,E2 -19492.21} C_VEL
LIN {X 0,Y 236.489,Z 209.071,A -85,B 0,C 180,E1 -19492.68,E2 -19492.68} C_VEL
LIN {X 0,Y 236.275,Z 211.985,A -85,B 0,C 180,E1 -19495.591,E2 -19495.591} C_VEL
LIN {X 0,Y 235.42,Z 215.889,A -85,B 0,C 180,E1 -19499.32,E2 -19499.32} C_VEL
LIN {X 0,Y 237.027,Z 221.901,A -85,B 0,C 180,E1 -19499.851,E2 -19499.851} C_VEL
LIN {X 0,Y 239.897,Z 233.529,A -85,B 0,C 180,E1 -19501.039,E2 -19501.039} C_VEL
LIN {X 0,Y 242,Z 245.453,A -85,B 0,C 180,E1 -19502.452,E2 -19502.452} C_VEL
LIN {X 0,Y 243.043,Z 255.693,A -85,B 0,C 180,E1 -19503.843,E2 -19503.843} C_VEL
LIN {X 0,Y 243.429,Z 267.431,A -85,B 0,C 180,E1 -19505.71,E2 -19505.71} C_VEL
LIN {X 0,Y 242.837,Z 272.373,A -85,B 0,C 180,E1 -19506.553,E2 -19506.553} C_VEL
LIN {X 0,Y 240.485,Z 282.866,A -85,B 0,C 180,E1 -19508.577,E2 -19508.577} C_VEL
LIN {X 0,Y 238.681,Z 291.296,A -85,B 0,C 180,E1 -19510.637,E2 -19510.637} C_VEL
LIN {X 0,Y 236.681,Z 299.65,A -85,B 0,C 180,E1 -19513.173,E2 -19513.173} C_VEL
LIN {X 0,Y 235.042,Z 306.324,A -85,B 0,C 180,E1 -19515.721,E2 -19515.721} C_VEL
LIN {X 0,Y 233.81,Z 312.433,A -85,B 0,C 180,E1 -19518.735,E2 -19518.735} C_VEL
LIN {X 0,Y 233.173,Z 316.403,A -85,B 0,C 180,E1 -19521.334,E2 -19521.334} C_VEL
LIN {X 0,Y 232.89,Z 318.444,A -85,B 0,C 180,E1 -19523.069,E2 -19523.069} C_VEL
LIN {X 0,Y 232.689,Z 320.514,A -85,B 0,C 180,E1 -19525.352,E2 -19525.352} C_VEL
LIN {X 0,Y 232.749,Z 322.077,A -85,B 0,C 180,E1 -19528.271,E2 -19528.271} C_VEL
LIN {X 0,Y 232.801,Z 322.454,A -85,B 0,C 180,E1 -19530.001,E2 -19530.001} C_VEL
LIN {X 0,Y 232.742,Z 322.441,A -85,B 0,C 180,E1 -19531.731,E2 -19531.731} C_VEL
LIN {X 0,Y 232.688,Z 321.516,A -85,B 0,C 180,E1 -19534.645,E2 -19534.645} C_VEL
LIN {X 0,Y 232.89,Z 319.985,A -85,B 0,C 180,E1 -19536.934,E2 -19536.934} C_VEL
LIN {X 0,Y 233.394,Z 317.365,A -85,B 0,C 180,E1 -19539.534,E2 -19539.534} C_VEL
LIN {X 0,Y 234.234,Z 313.738,A -85,B 0,C 180,E1 -19542.124,E2 -19542.124} C_VEL
LIN {X 0,Y 235.454,Z 309.007,A -85,B 0,C 180,E1 -19544.697,E2 -19544.697} C_VEL
LIN {X 0,Y 237.56,Z 301.914,A -85,B 0,C 180,E1 -19547.652,E2 -19547.652} C_VEL
LIN {X 0,Y 239.451,Z 295.084,A -85,B 0,C 180,E1 -19549.896,E2 -19549.896} C_VEL
LIN {X 0,Y 241.763,Z 286.354,A -85,B 0,C 180,E1 -19552.204,E2 -19552.204} C_VEL
LIN {X 0,Y 244.287,Z 276.764,A -85,B 0,C 180,E1 -19554.202,E2 -19554.202} C_VEL
LIN {X 0,Y 245.525,Z 271.143,A -85,B 0,C 180,E1 -19555.2,E2 -19555.2} C_VEL
LIN {X 0,Y 245.268,Z 260.338,A -85,B 0,C 180,E1 -19557.09,E2 -19557.09} C_VEL
LIN {X 0,Y 244.229,Z 249.411,A -85,B 0,C 180,E1 -19558.743,E2 -19558.743} C_VEL
LIN {X 0,Y 242.175,Z 237.605,A -85,B 0,C 180,E1 -19560.314,E2 -19560.314} C_VEL
LIN {X 0,Y 238.958,Z 224.93,A -85,B 0,C 180,E1 -19561.814,E2 -19561.814} C_VEL
LIN {X 0,Y 236.202,Z 216.18,A -85,B 0,C 180,E1 -19562.749,E2 -19562.749} C_VEL
LIN {X 0,Y 236.144,Z 215.683,A -85,B 0,C 180,E1 -19562.812,E2 -19562.812} C_VEL
LIN {X 0,Y 236.678,Z 213.052,A -85,B 0,C 180,E1 -19565.381,E2 -19565.381} C_VEL
LIN {X 0,Y 236.789,Z 209.974,A -85,B 0,C 180,E1 -19568.555,E2 -19568.555} C_VEL
LIN {X 0,Y 236.434,Z 206.897,A -85,B 0,C 180,E1 -19572.002,E2 -19572.002} C_VEL
LIN {X 0,Y 235.901,Z 203.828,A -85,B 0,C 180,E1 -19575.642,E2 -19575.642} C_VEL
LIN {X 0,Y 235.417,Z 201.236,A -85,B 0,C 180,E1 -19578.946,E2 -19578.946} C_VEL
LIN {X 0,Y 234.923,Z 198.226,A -85,B 0,C 180,E1 -19583.117,E2 -19583.117} C_VEL
LIN {X 0,Y 234.943,Z 198.224,A -85,B 0,C 180,E1 -19587.422,E2 -19587.422} C_VEL
LIN {X 0,Y 234.908,Z 198.227,A -85,B 0,C 180,E1 -19591.4,E2 -19591.4} C_VEL
LIN {X 0,Y 234.984,Z 198.215,A -85,B 0,C 180,E1 -19595.247,E2 -19595.247} C_VEL
LIN {X 0,Y 235.037,Z 198.208,A -85,B 0,C 180,E1 -19598.973,E2 -19598.973} C_VEL
LIN {X 0,Y 235.106,Z 198.199,A -85,B 0,C 180,E1 -19603.043,E2 -19603.043} C_VEL
LIN {X 0,Y 235.1,Z 198.198,A -85,B 0,C 180,E1 -19607.922,E2 -19607.922} C_VEL
LIN {X 0,Y 235.318,Z 198.172,A -85,B 0,C 180,E1 -19611.412,E2 -19611.412} C_VEL
LIN {X 0,Y 235.36,Z 198.167,A -85,B 0,C 180,E1 -19613.14,E2 -19613.14} C_VEL
LIN {X 0,Y 235.579,Z 198.14,A -85,B 0,C 180,E1 -19618.291,E2 -19618.291} C_VEL
LIN {X 0,Y 235.591,Z 198.138,A -85,B 0,C 180,E1 -19621.71,E2 -19621.71} C_VEL
LIN {X 0,Y 235.358,Z 198.166,A -85,B 0,C 180,E1 -19626.86,E2 -19626.86} C_VEL
LIN {X 0,Y 235.198,Z 198.188,A -85,B 0,C 180,E1 -19630.329,E2 -19630.329} C_VEL
LIN {X 0,Y 235.091,Z 198.201,A -85,B 0,C 180,E1 -19635.608,E2 -19635.608} C_VEL
LIN {X 0,Y 234.996,Z 198.214,A -85,B 0,C 180,E1 -19639.207,E2 -19639.207} C_VEL
LIN {X 0,Y 234.951,Z 198.218,A -85,B 0,C 180,E1 -19642.884,E2 -19642.884} C_VEL
LIN {X 0,Y 234.959,Z 198.216,A -85,B 0,C 180,E1 -19646.659,E2 -19646.659} C_VEL
LIN {X 0,Y 234.914,Z 198.222,A -85,B 0,C 180,E1 -19650.571,E2 -19650.571} C_VEL
LIN {X 0,Y 234.923,Z 198.223,A -85,B 0,C 180,E1 -19654.64,E2 -19654.64} C_VEL
LIN {X 0,Y 234.937,Z 198.221,A -85,B 0,C 180,E1 -19658.946,E2 -19658.946} C_VEL
LIN {X 0,Y 234.871,Z 198.228,A -85,B 0,C 180,E1 -19663.491,E2 -19663.491} C_VEL
